// TIA Portal V16 program export: 2 tag tables, 6 data types, 3 data blocks, 4 code blocks (in call order from the OBs), 0 instance data blocks

VAR_GLOBAL   // PLC tag table "Default tag table"
END_VAR

VAR_GLOBAL   // PLC tag table "PAL_SystemTags"
   _SysSignals01 AT %MB0 : Byte;   // System signals byte 01 — Logic and scan synchronised pulses   {ExternalWritable false}
   _False AT %M0.0 : Bool;   // System Logic Bit — Always FALSE   {ExternalWritable false}
   _True AT %M0.1 : Bool;   // System Logic Bit — Always TRUE   {ExternalWritable false}
   _50ms AT %M0.2 : Bool;   // System Timing — 50 ms pulse scan synchronised   {ExternalWritable false}
   _100ms AT %M0.3 : Bool;   // System Timing — 100 ms pulse scan synchronised   {ExternalWritable false}
   _200ms AT %M0.4 : Bool;   // System Timing — 200 ms pulse scan synchronised   {ExternalWritable false}
   _500ms AT %M0.5 : Bool;   // System Timing — 500 ms pulse scan synchronised   {ExternalWritable false}
   _1s AT %M0.6 : Bool;   // System Timing — 1 s pulse scan synchronised   {ExternalWritable false}
   _2s AT %M0.7 : Bool;   // System Timing — 2 s pulse scan synchronised   {ExternalWritable false}
   _SysSignals02 AT %MB1 : Byte;   // System signals byte 02 — scan signals and common square waves   {ExternalWritable false}
   _CycleTick AT %M1.0 : Bool;   // System Timing — Cycle tick (active odd cycles, alternates with _CycleTock)   {ExternalWritable false}
   _CycleTock AT %M1.1 : Bool;   // System Timing — Cycle tock (active even cycles, alternates with _CycleTick)   {ExternalWritable false}
   _CycleFirst AT %M1.2 : Bool;   // System Timing — First cycle detected   {ExternalWritable false}
   _100msSqW AT %M1.3 : Bool;   // System Timing — 100 ms square wave scan synchronised   {ExternalWritable false}
   _200msSqW AT %M1.4 : Bool;   // System Timing — 200 ms square wave scan synchronised   {ExternalWritable false}
   _500msSqW AT %M1.5 : Bool;   // System Timing — 500 ms square wave scan synchronised   {ExternalWritable false}
   _1sSqW AT %M1.6 : Bool;   // System Timing — 1 s square wave scan synchronised   {ExternalWritable false}
   _2sSqW AT %M1.7 : Bool;   // System Timing — 2 s square wave scan synchronised   {ExternalWritable false}
   _ClockMem AT %MB10 : Byte;   // Clock Memory (populated by the CPU)   {ExternalWritable false}
   _ClockMem_100msSqW AT %M10.0 : Bool;   // Clock Memory — 10.0 Hz square wave 0.1 s period   {ExternalWritable false}
   _ClockMem_200msSqW AT %M10.1 : Bool;   // Clock Memory — 5.00 Hz square wave 0.2 s period   {ExternalWritable false}
   _ClockMem_400msSqW AT %M10.2 : Bool;   // Clock Memory — 2.50 Hz square wave 0.4 s period   {ExternalWritable false}
   _ClockMem_500msSqW AT %M10.3 : Bool;   // Clock Memory — 2.00 Hz square wave 0.5 s period   {ExternalWritable false}
   _ClockMem_800msSqW AT %M10.4 : Bool;   // Clock Memory — 1.25 Hz square wave 0.8 s period   {ExternalWritable false}
   _ClockMem_1000msSqW AT %M10.5 : Bool;   // Clock Memory — 1.00 Hz square wave 1.0 s period   {ExternalWritable false}
   _ClockMem_1600msSqW AT %M10.6 : Bool;   // Clock Memory — 0.62 Hz square wave 1.6 s period   {ExternalWritable false}
   _ClockMem_2000msSqW AT %M10.7 : Bool;   // Clock Memory — 0.50 Hz square wave 2.0 s period   {ExternalWritable false}
   _SysSignals AT %MW0 : Int;   // System signals   {ExternalWritable false}
END_VAR

TYPE "UT01000_St_SysRevision"
TITLE = Static UDT — Sys - Revision Data
// Revision Data
// stored: IsFailsafeCompliant false
   STRUCT
      REV_BLOCK { ExternalWritable := 'False'; S7_SetPoint := 'True'} : String[7];   // Block or Project number
      REV_NUMBER { ExternalWritable := 'False'; S7_SetPoint := 'True'} : String[20];   // Revision status followed by revision number
      REV_DATE { ExternalWritable := 'False'; S7_SetPoint := 'True'} : String[10];   // Revision date
      REV_AUTHOR { ExternalWritable := 'False'; S7_SetPoint := 'True'} : String[20];   // Revision author
   END_STRUCT;
END_TYPE

TYPE "UT01001_St_SysLicence"
TITLE = Static UDT — Sys - Licence Information
// Licence Information
// stored: IsFailsafeCompliant false
   STRUCT
      LICENCE_TYPE { ExternalWritable := 'False'} : String[20];   // Licence information — type of licence
      COPYRIGHT { ExternalWritable := 'False'} : String[30];   // Licence information — copyright (year and name)
   END_STRUCT;
END_TYPE

TYPE "UT21000_Dy_SysSignals"
TITLE = Dynamic UDT — Sys - Global Signals
// Global Logic and Timing Signals
// stored: IsFailsafeCompliant false
   STRUCT
      revInfo { ExternalWritable := 'False'} : "UT01000_St_SysRevision";   // ▀▀▀▀ UDT CURRENT REVISION
      ___________0010_0 { ExternalAccessible := 'False'; ExternalVisible := 'False'; ExternalWritable := 'False'} : Bool;
      ___________0010_1 { ExternalAccessible := 'False'; ExternalVisible := 'False'; ExternalWritable := 'False'} : Bool;   // ▀▀▀▀ SYSTEM SIGNALS
      _False { ExternalWritable := 'False'} : Bool;   // System Logic Bit — Always FALSE
      _True { ExternalWritable := 'False'} : Bool;   // System Logic Bit — Always TRUE
      _50ms { ExternalWritable := 'False'} : Bool;   // System Timing — 50 ms Pulse Scan synchronised
      _100ms { ExternalWritable := 'False'} : Bool;   // System Timing — 100 ms Pulse Scan synchronised
      _200ms { ExternalWritable := 'False'} : Bool;   // System Timing — 200 ms Pulse Scan synchronised
      _500ms { ExternalWritable := 'False'} : Bool;   // System Timing — 500 ms Pulse Scan synchronised
      _1s { ExternalWritable := 'False'} : Bool;   // System Timing — 1 s Pulse Scan synchronised
      _2s { ExternalWritable := 'False'} : Bool;   // System Timing — 2 s Pulse Scan synchronised
      _CycleTick { ExternalWritable := 'False'} : Bool;   // System Timing — Cycle tick (active odd cycles, alternates with _CycleTock)
      _CycleTock { ExternalWritable := 'False'} : Bool;   // System Timing — Cycle tock (active even cycles, alternates with _CycleTick)
      _CycleFirst { ExternalWritable := 'False'} : Bool;   // System Timing — First cycle detected
      _100msSqW { ExternalWritable := 'False'} : Bool;   // System Timing — 100 ms Square wave Scan synchronised
      _200msSqW { ExternalWritable := 'False'} : Bool;   // System Timing — 200 ms Square wave Scan synchronised
      _500msSqW { ExternalWritable := 'False'} : Bool;   // System Timing — 500 ms Square wave Scan synchronised
      _1sSqW { ExternalWritable := 'False'} : Bool;   // System Timing — 1 s Square wave Scan synchronised
      _2sSqW { ExternalWritable := 'False'} : Bool;   // System Timing — 2 s Square wave Scan synchronised
   END_STRUCT;
   // revInfo.REV_BLOCK := 'UT21000';
   // revInfo.REV_NUMBER := '000-801';
   // revInfo.REV_DATE := '2021-02-18';
   // revInfo.REV_AUTHOR := 'M. Gledhill';
END_TYPE

TYPE "UT21001_Dy_SysData"
TITLE = Dynamic UDT — Sys - Global Data
// Global System Data
// stored: IsFailsafeCompliant false
   STRUCT
      revInfo { ExternalWritable := 'False'} : "UT01000_St_SysRevision";   // ▀▀▀▀ UDT CURRENT REVISION
      ___________0010_0 { ExternalAccessible := 'False'; ExternalVisible := 'False'; ExternalWritable := 'False'} : Bool;
      ___________0010_1 { ExternalAccessible := 'False'; ExternalVisible := 'False'; ExternalWritable := 'False'} : Bool;   // ▀▀▀▀ CYCLE TIME DATA
      CycTime_Prev { ExternalWritable := 'False'} : Real;   // Previous cycle time (ms)
      CycTime_Max { ExternalWritable := 'False'} : Real;   // Maximum cycle time - since start-up (ms)
      CycTime_Min { ExternalWritable := 'False'} : Real;   // Minimum cycle time - since start-up (ms)
      Cyc_Counter { ExternalWritable := 'False'} : UDInt;   // Cycle rolling counter - incremented by 1 each scan
      __________0020_0 { ExternalAccessible := 'False'; ExternalVisible := 'False'; ExternalWritable := 'False'} : Bool := false;
      __________0020_1 { ExternalAccessible := 'False'; ExternalVisible := 'False'; ExternalWritable := 'False'} : Bool := false;   // ▀▀▀▀ REAL TIME CLOCK DATA
      RTC_Year { ExternalWritable := 'False'} : Int;   // Year (returns a value in the range 1970 to 2262)
      RTC_Month { ExternalWritable := 'False'} : Int;   // Month (1-12 representing Jan to Dec)
      RTC_Day { ExternalWritable := 'False'} : Int;   // Day of month (1-31)
      RTC_DayofWeek { ExternalWritable := 'False'} : Int;   // Day of week (1-7, where 1=Sunday, 7=Saturday)
      RTC_Hour { ExternalWritable := 'False'} : Int;   // Hour of day (0-23)
      RTC_Minute { ExternalWritable := 'False'} : Int;   // Minutes (0-59)
      RTC_Second { ExternalWritable := 'False'} : Int;   // Seconds (0-59)
      RTC_millisecond { ExternalWritable := 'False'} : Int;   // Milliseconds (0-999)
   END_STRUCT;
   // revInfo.REV_BLOCK := 'UT21001';
   // revInfo.REV_NUMBER := '001.000';
   // revInfo.REV_DATE := '2021-02-18';
   // revInfo.REV_AUTHOR := 'M. Gledhill ';
END_TYPE

TYPE "UT02001_St_InstAnalogRead"
TITLE = Static UDT — Inst - Analogue Instrument Read and Scale
// Analogue Instrument Read and Scale
// stored: IsFailsafeCompliant false
   STRUCT
      revInfo { ExternalWritable := 'False'} : "UT01000_St_SysRevision";   // Revision information
      ___________0010_0 { ExternalAccessible := 'False'; ExternalVisible := 'False'; ExternalWritable := 'False'} : Int;
      ___________0010_1 { ExternalAccessible := 'False'; ExternalVisible := 'False'; ExternalWritable := 'False'} : Int;   // ▀▀▀▀ INSTRUMENT CONFIGURATION
      CONFIG_ALM_H_ENABLE { ExternalWritable := 'False'; S7_SetPoint := 'True'} : Bool;   // CONFIG — High alarm is enabled (1 = enabled, 0 = no alarm)
      CONFIG_ALM_L_ENABLE { ExternalWritable := 'False'; S7_SetPoint := 'True'} : Bool;   // CONFIG — Low alarm is enabled (1 = enabled, 0 = no alarm)
      CONFIG_WRN_H_ENABLE { ExternalWritable := 'False'; S7_SetPoint := 'True'} : Bool;   // CONFIG — High warning is enabled (1 = enabled, 0 = no warning)
      CONFIG_WRN_L_ENABLE { ExternalWritable := 'False'; S7_SetPoint := 'True'} : Bool;   // CONFIG — Low warning is enabled (1 = enabled, 0 = no warning)
      CONFIG_FP_DISABLE { ExternalWritable := 'False'; S7_SetPoint := 'True'} : Bool;   // CONFIG — Faceplate is disabled (1 = no Faceplate, 0 = normal)
      CONFIG_SIM_DISABLE { ExternalWritable := 'False'; S7_SetPoint := 'True'} : Bool;   // CONFIG — Simulation is disabled (1 = no Simulation, 0 = normal)
      CONFIG_RL_ENABLE { ExternalWritable := 'False'; S7_SetPoint := 'True'} : Bool;   // CONFIG — Remote/local mode enabled (1 = remote/local permitted, 0 = remote/local N/A)
      ___________0020_0 { ExternalAccessible := 'False'; ExternalVisible := 'False'; ExternalWritable := 'False'} : Int;
      ___________0020_1 { ExternalAccessible := 'False'; ExternalVisible := 'False'; ExternalWritable := 'False'} : Int;   // ▀▀▀▀ INSTRUMENT RANGE & SCALING DATA
      RANGE_RAW_MIN { ExternalWritable := 'False'; S7_SetPoint := 'True'} : Int;   // RANGE — Minimum value of the raw analogue signal (at the card)
      RANGE_RAW_MAX { ExternalWritable := 'False'; S7_SetPoint := 'True'} : Int;   // RANGE — Maximum value of the raw analogue signal (at the card)
      RANGE_SCALE_MIN { ExternalWritable := 'False'; S7_SetPoint := 'True'} : Real;   // RANGE — Minimum value of the scaled analogue signal [engineering units]
      RANGE_SCALE_MAX { ExternalWritable := 'False'; S7_SetPoint := 'True'} : Real;   // RANGE — Maximum value of the scaled analogue signal [engineering units]
      RANGE_OOR_PERCENT { ExternalWritable := 'False'; S7_SetPoint := 'True'} : Real;   // RANGE — Out of range percentage (of raw range), beyond which the instrument is out of range
      ___________0030_0 { ExternalAccessible := 'False'; ExternalVisible := 'False'; ExternalWritable := 'False'} : Int;
      ___________0030_1 { ExternalAccessible := 'False'; ExternalVisible := 'False'; ExternalWritable := 'False'} : Int;   // ▀▀▀▀ INSTRUMENT INFORMATION (TAG & UNITS)
      INFO_TAG { ExternalWritable := 'False'; S7_SetPoint := 'True'} : String[20];   // INFORMATION — Instrument ID tag
      INFO_UNITS { ExternalWritable := 'False'; S7_SetPoint := 'True'} : String[10];   // INFORMATION — Engineering units of the instrument (unit of measure)
      ___________0040_0 { ExternalAccessible := 'False'; ExternalVisible := 'False'; ExternalWritable := 'False'} : Int;
      ___________0040_1 { ExternalAccessible := 'False'; ExternalVisible := 'False'; ExternalWritable := 'False'} : Int;   // ▀▀▀▀ INSTRUMENT ALARM/WARNING & HYSTERESIS SETPOINTS
      SP_ALM_H_VAL { ExternalWritable := 'False'; S7_SetPoint := 'True'} : Real;   // SETPOINT — High alarm threshold value [engineering units]
      SP_ALM_L_VAL { ExternalWritable := 'False'; S7_SetPoint := 'True'} : Real;   // SETPOINT — Low alarm threshold value [engineering units]
      SP_WRN_H_VAL { ExternalWritable := 'False'; S7_SetPoint := 'True'} : Real;   // SETPOINT — High warning threshold value [engineering units]
      SP_WRN_L_VAL { ExternalWritable := 'False'; S7_SetPoint := 'True'} : Real;   // SETPOINT — Low warning threshold value [engineering units]
      SP_ALM_H_HYST_VAL { ExternalWritable := 'False'; S7_SetPoint := 'True'} : Real;   // SETPOINT — High alarm hysteresis value [engineering units]
      SP_ALM_L_HYST_VAL { ExternalWritable := 'False'; S7_SetPoint := 'True'} : Real;   // SETPOINT — Low alarm hysteresis value [engineering units]
      SP_WRN_H_HYST_VAL { ExternalWritable := 'False'; S7_SetPoint := 'True'} : Real;   // SETPOINT — High warning hysteresis value [engineering units]
      SP_WRN_L_HYST_VAL { ExternalWritable := 'False'; S7_SetPoint := 'True'} : Real;   // SETPOINT — Low warning hysteresis value [engineering units]
      ___________0050_0 { ExternalAccessible := 'False'; ExternalVisible := 'False'; ExternalWritable := 'False'} : Int;
      ___________0050_1 { ExternalAccessible := 'False'; ExternalVisible := 'False'; ExternalWritable := 'False'} : Int;   // ▀▀▀▀ INSTRUMENT TIMER DEFAULT VALUES
      TIME_ALM_H_ON_DEL { ExternalWritable := 'False'; S7_SetPoint := 'True'} : Real;   // TIMER — High alarm on delay time (activation delay), [seconds]
      TIME_ALM_L_ON_DEL { ExternalWritable := 'False'; S7_SetPoint := 'True'} : Real;   // TIMER — Low alarm on delay time (activation delay), [seconds]
      TIME_WRN_H_ON_DEL { ExternalWritable := 'False'; S7_SetPoint := 'True'} : Real;   // TIMER — High warning on delay time (activation delay), [seconds]
      TIME_WRN_L_ON_DEL { ExternalWritable := 'False'; S7_SetPoint := 'True'} : Real;   // TIMER — Low warning on delay time (activation delay), [seconds]
      TIME_ALM_H_OFF_DEL { ExternalWritable := 'False'; S7_SetPoint := 'True'} : Real;   // TIMER — High alarm off delay time (deactivation delay), [seconds]
      TIME_ALM_L_OFF_DEL { ExternalWritable := 'False'; S7_SetPoint := 'True'} : Real;   // TIMER — Low alarm off delay time (deactivation delay), [seconds]
      TIME_WRN_H_OFF_DEL { ExternalWritable := 'False'; S7_SetPoint := 'True'} : Real;   // TIMER — High warning off delay time (deactivation delay), [seconds]
      TIME_WRN_L_OFF_DEL { ExternalWritable := 'False'; S7_SetPoint := 'True'} : Real;   // TIMER — Low warning off delay time (deactivation delay), [seconds]
   END_STRUCT;
   // revInfo.REV_BLOCK := 'UT02001';
   // revInfo.REV_NUMBER := '001.000';
   // revInfo.REV_DATE := '2021-02-18';
   // revInfo.REV_AUTHOR := 'M. Gledhill ';
END_TYPE

TYPE "UT22001_Dy_InstAnalogRead"
TITLE = Dynamic UDT — Inst - Analogue Instrument Read and Scale
// Analogue Instrument Read and Scale
// stored: IsFailsafeCompliant false
   STRUCT
      revInfo : "UT01000_St_SysRevision";   // Revision information
      ___________0010_0 { ExternalAccessible := 'False'; ExternalVisible := 'False'; ExternalWritable := 'False'} : Int;
      ___________0010_1 { ExternalAccessible := 'False'; ExternalVisible := 'False'; ExternalWritable := 'False'} : Int;   // ▀▀▀▀ STATUS (FOR BLOCK ICON AND SYMBOL)
      status_ConfigError : Bool;   // STATUS — Block is configured incorrectly
      status_Alm_H : Bool;   // STATUS — High alarm is active (1 = alarm active, 0 = no alarm)
      status_Alm_L : Bool;   // STATUS — Low alarm is active (1 = alarm active, 0 = no alarm)
      status_Wrn_H : Bool;   // STATUS — High warning is active (1 = warning active, 0 = no warning)
      status_Wrn_L : Bool;   // STATUS — Low warning is active (1 = warning active, 0 = no warning)
      status_Alm_H_Mask : Bool;   // STATUS — High alarm is masked (1 = alarm masked, 0 = normal)
      status_Alm_L_Mask : Bool;   // STATUS — Low alarm is masked (1 = alarm masked, 0 = normal)
      status_Wrn_H_Mask : Bool;   // STATUS — High warning is masked (1 = warning masked, 0 = normal)
      status_Wrn_L_Mask : Bool;   // STATUS — Low warning is masked (1 = warning masked, 0 = normal)
      status_Alm_H_Dis : Bool;   // STATUS — High alarm is disabled (1 = alarm disabled, 0 = normal)
      status_Alm_L_Dis : Bool;   // STATUS — Low alarm is disabled (1 = alarm disabled, 0 = normal)
      status_Wrn_H_Dis : Bool;   // STATUS — High warning is disabled (1 = warning disabled, 0 = normal)
      status_Wrn_L_Dis : Bool;   // STATUS — Low warning is disabled (1 = warning disabled, 0 = normal)
      status_Fault : Bool;   // STATUS — Instrument is in fault (1 = fault present, 0 = healthy)
      status_SimOn : Bool;   // STATUS — Instrument is in simulation mode (1 = simulation mode on, 0 = normal)
      status_RemoteOn : Bool;   // STATUS — Instrument is in remote mode (1 = remote mode, 0 = remote mode off)
      status_LocalOn : Bool;   // STATUS — Instrument is in local mode (1 = local mode, 0 = local mode off)
      status_RLOff : Bool;   // STATUS — Remote/local mode disabled (1 = ALL mode on, 0 = RL mode selected)
      ___________0020_0 { ExternalAccessible := 'False'; ExternalVisible := 'False'; ExternalWritable := 'False'} : Int;
      ___________0020_1 { ExternalAccessible := 'False'; ExternalVisible := 'False'; ExternalWritable := 'False'} : Int;   // ▀▀▀▀ OPERATING MODE SELECTION (FROM FACEPLATE OR PANEL)
      mode_Alm_H_MaskOn : Bool;   // MODE — Mask Alm_H (1 = mask alarm, 0 = normal)
      mode_Alm_L_MaskOn : Bool;   // MODE — Mask Alm_L (1 = mask alarm, 0 = normal)
      mode_Wrn_H_MaskOn : Bool;   // MODE — Mask Wrn_H (1 = mask warning, 0 = normal)
      mode_Wrn_L_MaskOn : Bool;   // MODE — Mask Wrn_H (1 = mask warning, 0 = normal)
      mode_SimOn : Bool;   // MODE — Simulation mode (1 = simulation mode active, 0 = normal)
      mode_SimValue : Real;   // MODE — Simulation value [engineering units]
      mode_LocalOn : Bool;   // MODE — Local HMI control enabled (1 = control active, 0 = control disabled or N/A)
      mode_RemoteOn : Bool;   // MODE — Remote SCADA control enabled (1 = control active, 0 = control disabled or N/A)
      ___________0030_0 { ExternalAccessible := 'False'; ExternalVisible := 'False'; ExternalWritable := 'False'} : Int;
      ___________0030_1 { ExternalAccessible := 'False'; ExternalVisible := 'False'; ExternalWritable := 'False'} : Int;   // ▀▀▀▀ MESSAGES (ALARMS, WARNINGS, FAULTS AND EVENTS)
      msg_Alm_H : Bool;   // MESSAGE — Alarm - high alarm is active
      msg_Alm_L : Bool;   // MESSAGE — Alarm - low alarm is active
      msg_Wrn_H : Bool;   // MESSAGE — Warning - high warning is active
      msg_Wrn_L : Bool;   // MESSAGE — Warning - low warning is active
      msg_Flt_External : Bool;   // MESSAGE — Fault - external fault signal is active
      msg_Flt_OverRange : Bool;   // MESSAGE — Fault - instrument is over-range
      msg_Flt_UnderRange : Bool;   // MESSAGE — Fault - instrument is under-range
      msg_Flt_OutOfRange : Bool;   // MESSAGE — Fault - instrument is out-of-range
      ___________0040_0 { ExternalAccessible := 'False'; ExternalVisible := 'False'; ExternalWritable := 'False'} : Int;
      ___________0040_1 { ExternalAccessible := 'False'; ExternalVisible := 'False'; ExternalWritable := 'False'} : Int;   // ▀▀▀▀ BATCH AND BOOKING DATA
      batch_ID : Int;   // BATCH — Booking ID (optional for batch operations)
      ___________0050_0 { ExternalAccessible := 'False'; ExternalVisible := 'False'; ExternalWritable := 'False'} : Int;
      ___________0050_1 { ExternalAccessible := 'False'; ExternalVisible := 'False'; ExternalWritable := 'False'} : Int;   // ▀▀▀▀ LIVE DATA (SCALED READING & TIMER VALUES)
      actual_Value : Real;   // ACTUAL — SCALED INSTRUMENT VALUE [engineering units]
      actual_Alm_H_Timer : Real;   // ACTUAL — Timer value — alarm high operation timer [seconds]
      actual_Alm_L_Timer : Real;   // ACTUAL — Timer value — alarm low operation timer [seconds]
      actual_Wrn_H_Timer : Real;   // ACTUAL — Timer value — warning high operation timer [seconds]
      actual_Wrn_L_Timer : Real;   // ACTUAL — Timer value — warning low operation timer [seconds]
      ___________0090_0 { ExternalAccessible := 'False'; ExternalVisible := 'False'; ExternalWritable := 'False'} : Int;
      ___________0090_1 { ExternalAccessible := 'False'; ExternalVisible := 'False'; ExternalWritable := 'False'} : Int;   // ▀▀▀▀ BLOCK INTERNAL WORKING AND STORAGE AREA
      "$pret_AlmHEn" : Bool;   // INTERNAL — Edge retention (+ve) alarm high enable
      "$Pret_AlmLEn" : Bool;   // INTERNAL — Edge retention (+ve) alarm low enable
      "$pret_WrnHEn" : Bool;   // INTERNAL — Edge retention (+ve) warning high enable
      "$pret_WrnLEn" : Bool;   // INTERNAL — Edge retention (+ve) warning low enable
   END_STRUCT;
   // revInfo.REV_BLOCK := 'UT22001';
   // revInfo.REV_NUMBER := '000.801';
   // revInfo.REV_DATE := '2021-02-18';
   // revInfo.REV_AUTHOR := 'M. Gledhill';
END_TYPE

DATA_BLOCK "DB21001_Dy_SysGlobalData"   // DB21001
TITLE = Dynamic DB — Sys - Global Data
{ S7_Optimized_Access := 'TRUE' }
AUTHOR : M_Gledhill
FAMILY : System
NAME : Dy_SysGlobalData
VERSION : 1.0
// PRACTICAL SERIES AUTOMATION LIBRARY (PAL)   —   COPYRIGHT 2020 – M. GLEDHILL (MIT LICENCE)
//                   ———— ◆ ————
//  FOR DETAILED DOCUMENTATION — SELECT THE BLOCK IN THE PROJECT TREE AND PRESS SHIFT + F1
//  FULL ONLINE DOCUMENTATION IS AVAILABLE AT: https://practicalseries.com/2001-pal/index.html
// stored: AutoNumber false, DBAccessibleFromOPCUA true, IsOnlyStoredInLoadMemory false, IsRetainMemResEnabled false, IsWriteProtectedInAS false, MemoryReserve 100
   VAR
      _DB_Header { ExternalWritable := 'False'} : Array[0..79] of Bool;   // STANDARD SYSTEM GLOBAL DATA
      __________0000_0 { ExternalWritable := 'False'} : Bool := false;
      __________0000_1 { ExternalWritable := 'False'} : Bool := false;   // ▀▀▀▀ DB CURRENT REVISION
      revInfo { ExternalWritable := 'False'} : "UT01000_St_SysRevision";
      __________0010_0 { ExternalWritable := 'False'} : Bool := false;
      __________0010_1 { ExternalWritable := 'False'} : Bool := false;   // ▀▀▀▀ PROJECT CURRENT REVISION
      projRevInfo { ExternalWritable := 'False'} : "UT01000_St_SysRevision";
      __________0020_0 { ExternalWritable := 'False'} : Bool := false;
      __________0020_1 { ExternalWritable := 'False'} : Bool := false;   // ▀▀▀▀ SYSTEM SIGNALS — LOGIC AND TIMING SIGNALS
      SysSignals { ExternalWritable := 'False'} : "UT21000_Dy_SysSignals";
      __________0030_0 { ExternalWritable := 'False'} : Bool := false;
      __________0030_1 { ExternalWritable := 'False'} : Bool := false;   // ▀▀▀▀ SYSTEM DATA — CYCLE TIMING AND RTC
      SysData { ExternalWritable := 'False'} : "UT21001_Dy_SysData";
      __________0040_0 { ExternalWritable := 'False'} : Bool := false;
      __________0040_1 { ExternalWritable := 'False'} : Bool := false;   // ▀▀▀▀ OB CALL TIMES
      OB10_CallTime { ExternalWritable := 'False'} : DTL;   // Time of day interrupt 1
      OB11_CallTime { ExternalWritable := 'False'} : DTL;   // Time of day interrupt 2
      OB12_CallTime { ExternalWritable := 'False'} : DTL;   // Time of day interrupt 3
      OB13_CallTime { ExternalWritable := 'False'} : DTL;   // Time of day interrupt 4
      OB14_CallTime { ExternalWritable := 'False'} : DTL;   // Time of day interrupt 5
      OB15_CallTime { ExternalWritable := 'False'} : DTL;   // Time of day interrupt 6
      OB16_CallTime { ExternalWritable := 'False'} : DTL;   // Time of day interrupt 7
      OB17_CallTime { ExternalWritable := 'False'} : DTL;   // Time of day interrupt 8
      OB20_CallTime { ExternalWritable := 'False'} : DTL;   // Time delay interrupt 1
      OB21_CallTime { ExternalWritable := 'False'} : DTL;   // Time delay interrupt 2
      OB22_CallTime { ExternalWritable := 'False'} : DTL;   // Time delay interrupt 3
      OB23_CallTime { ExternalWritable := 'False'} : DTL;   // Time delay interrupt 4
      OB30_CallTime { ExternalWritable := 'False'} : DTL;   // Timed cyclic interrupt 1
      OB31_CallTime { ExternalWritable := 'False'} : DTL;   // Timed cyclic interrupt 2
      OB32_CallTime { ExternalWritable := 'False'} : DTL;   // Timed cyclic interrupt 3
      OB33_CallTime { ExternalWritable := 'False'} : DTL;   // Timed cyclic interrupt 4
      OB34_CallTime { ExternalWritable := 'False'} : DTL;   // Timed cyclic interrupt 5
      OB35_CallTime { ExternalWritable := 'False'} : DTL;   // Timed cyclic interrupt 6
      OB36_CallTime { ExternalWritable := 'False'} : DTL;   // Timed cyclic interrupt 7
      OB37_CallTime { ExternalWritable := 'False'} : DTL;   // Timed cyclic interrupt 8
      OB38_CallTime { ExternalWritable := 'False'} : DTL;   // Timed cyclic interrupt 9
      OB40_CallTime { ExternalWritable := 'False'} : DTL;   // Hardware interrupt 1
      OB41_CallTime { ExternalWritable := 'False'} : DTL;   // Hardware interrupt 2
      OB42_CallTime { ExternalWritable := 'False'} : DTL;   // Hardware interrupt 3
      OB43_CallTime { ExternalWritable := 'False'} : DTL;   // Hardware interrupt 4
      OB44_CallTime { ExternalWritable := 'False'} : DTL;   // Hardware interrupt 5
      OB45_CallTime { ExternalWritable := 'False'} : DTL;   // Hardware interrupt 6
      OB46_CallTime { ExternalWritable := 'False'} : DTL;   // Hardware interrupt 7
      OB47_CallTime { ExternalWritable := 'False'} : DTL;   // Hardware interrupt 8
      OB80_CallTime { ExternalWritable := 'False'} : DTL;   // Error interrupt — max cycle time exceeded
      OB82_CallTime { ExternalWritable := 'False'} : DTL;   // Error interrupt — module diagnostic
      OB83_CallTime { ExternalWritable := 'False'} : DTL;   // Error interrupt — module changed
      OB86_CallTime { ExternalWritable := 'False'} : DTL;   // Error interrupt — rack fault
      OB100_CallTime { ExternalWritable := 'False'} : DTL;   // Start-up interrupt
      OB121_CallTime { ExternalWritable := 'False'} : DTL;   // Error interrupt — programming fault
      OB122_CallTime { ExternalWritable := 'False'} : DTL;   // Error interrupt — IO access fault
   END_VAR
BEGIN
   // _DB_Header[0] : ▀▀▀▀▀▀▀▀▀▀▀▀▀▀▀▀▀▀▀▀▀▀▀▀▀▀▀▀▀▀▀▀▀▀▀▀▀▀▀▀▀▀▀▀
   // _DB_Header[2] : TITLE: STANDARD SYSTEM GLOBAL DATA
   // _DB_Header[4] : ▄▄▄▄▄▄▄▄▄▄▄▄▄▄▄▄▄▄▄▄▄▄▄▄▄▄▄▄▄▄▄▄▄▄▄▄▄▄▄▄▄▄▄▄
   // _DB_Header[5] : TYPE: DYNAMIC
   // _DB_Header[6] : ▀▀▀▀▀▀▀▀▀▀▀▀▀▀▀▀▀▀▀▀▀▀▀▀▀▀▀▀▀▀▀▀▀▀▀▀▀▀▀▀▀▀▀▀
   // _DB_Header[8] : Global system data storage DB. The block records various system variables and information:
   // _DB_Header[10] : • Project revision data
   // _DB_Header[11] : • Common system signals (logic and timing)
   // _DB_Header[12] : • Cycle timing information (previous, max, min and a cycle counter)
   // _DB_Header[13] : • CPU real time clock data (in globally readable format)
   // _DB_Header[14] : • Last call time of any interrupt OB
   // _DB_Header[16] : The cycle timing information and the RTC data are provided by FC01000. The interrupt OB data
   // _DB_Header[17] : is provided by the individual OBs.
   // _DB_Header[19] : ━━━ ⬙⬙⬙⬙⬙⬙ ━━━
   // _DB_Header[21] : ▄▄▄▄▄▄▄▄▄▄▄▄▄▄▄▄▄▄▄▄▄▄▄▄▄▄▄▄▄▄▄▄▄▄▄▄▄▄▄▄▄▄▄▄
   // _DB_Header[22] : MODIFICATION HISTORY
   // _DB_Header[24] : This is a summary of the recent software modifications made to this block (most recent at top)
   // _DB_Header[26] : ―――――――――――――――――――――――――――――――――――――――――――
   // _DB_Header[27] : DATE REVISION MASTER BRANCH DEV
   // _DB_Header[28] : (nnn.amm) COMMIT TAG (Base ---> Merge) BRANCH Author
   // _DB_Header[29] : ———————————————————————————————————————————
   // _DB_Header[30] : 2020.11.18 001.000 D0002A-001.000 D0002 D0003 D0002A M. Gledhill
   // _DB_Header[31] : FC01001 Migration to VCS — Released for use
   // _DB_Header[32] : 2020.11.18 000.801 D0002A-000.801 D0002 N/A D0002A M. Gledhill
   // _DB_Header[33] : FC01001 Migration to VCS — Released for test
   // _DB_Header[34] : ———————————————————————————————————————————
   // _DB_Header[35] : Where: nnn = Major revision
   // _DB_Header[36] : a = Type (1-7 Development, 8 Proving, 9 Qualification, 0 Release)
   // _DB_Header[37] : mm = Minor revision (must be 00 if a = 0)
   // _DB_Header[38] : Block properties version number should be set to nn.a (only one decimal place)
   // _DB_Header[40] : ██████████████ █ █ █ █ END █ █ █ █ ██████████████
   revInfo.REV_BLOCK := 'DB21001';
   revInfo.REV_NUMBER := '001.000';
   revInfo.REV_DATE := '2021-02-18';
   revInfo.REV_AUTHOR := 'M. Gledhill';
END_DATA_BLOCK

DATA_BLOCK "DB02001_St_InstAnalogRead"   // DB2001
TITLE = Static DB — Inst - Analogue Instrument Read and Scale
{ S7_Optimized_Access := 'TRUE' }
AUTHOR : M_Gledhill
FAMILY : Instrumentation
NAME : St_InstAnalogRead
VERSION : 1.0
// PRACTICAL SERIES AUTOMATION LIBRARY (PAL)   —   COPYRIGHT 2020 – M. GLEDHILL (MIT LICENCE)
//                   ———— ◆ ————
//  FOR DETAILED DOCUMENTATION — SELECT THE BLOCK IN THE PROJECT TREE AND PRESS SHIFT + F1
//  FULL ONLINE DOCUMENTATION IS AVAILABLE AT: https://practicalseries.com/2001-pal/index.html
// stored: AutoNumber false, DBAccessibleFromOPCUA true, IsOnlyStoredInLoadMemory false, IsRetainMemResEnabled false, IsWriteProtectedInAS false, MemoryReserve 100
   VAR
      _DB_Header { ExternalAccessible := 'False'; ExternalVisible := 'False'; ExternalWritable := 'False'} : Array[0..79] of Bool;   // STANDARD ANALOGUE INSTRUMENT READ
      __________0000_0 { ExternalAccessible := 'False'; ExternalVisible := 'False'; ExternalWritable := 'False'} : Bool := false;
      __________0000_1 { ExternalAccessible := 'False'; ExternalVisible := 'False'; ExternalWritable := 'False'} : Bool := false;   // ▀▀▀▀ DB CURRENT REVISION
      revInfo { ExternalWritable := 'False'; S7_SetPoint := 'True'} : "UT01000_St_SysRevision";
      __________0010_0 { ExternalAccessible := 'False'; ExternalVisible := 'False'; ExternalWritable := 'False'} : Bool := false;
      __________0010_1 { ExternalAccessible := 'False'; ExternalVisible := 'False'; ExternalWritable := 'False'} : Bool := false;   // ▀▀▀▀ ANALOGUE INSTRUMENTS
      FIC101 { ExternalWritable := 'False'; S7_SetPoint := 'True'} : "UT02001_St_InstAnalogRead";   // Filter 1 outlet flow
   END_VAR
BEGIN
   // _DB_Header[0] : ▀▀▀▀▀▀▀▀▀▀▀▀▀▀▀▀▀▀▀▀▀▀▀▀▀▀▀▀▀▀▀▀▀▀▀▀▀▀▀▀▀▀▀▀
   // _DB_Header[2] : TITLE: STANDARD ANALOGUE INSTRUMENT READ (SCALE & ALARM MONITORING)
   // _DB_Header[4] : ▄▄▄▄▄▄▄▄▄▄▄▄▄▄▄▄▄▄▄▄▄▄▄▄▄▄▄▄▄▄▄▄▄▄▄▄▄▄▄▄▄▄▄▄
   // _DB_Header[5] : TYPE: STATIC
   // _DB_Header[6] : ▀▀▀▀▀▀▀▀▀▀▀▀▀▀▀▀▀▀▀▀▀▀▀▀▀▀▀▀▀▀▀▀▀▀▀▀▀▀▀▀▀▀▀▀
   // _DB_Header[8] : This is the static data block associated with the standard analogue instrument read
   // _DB_Header[9] : block:
   // _DB_Header[10] : FC02001_StdInstAnalogRead
   // _DB_Header[12] : The static data holds the threshold values for any configured alarms and warnings,
   // _DB_Header[13] : activation delays, scaled and raw value ranges and various configuration options.
   // _DB_Header[15] : Each instrument is given the user data type:
   // _DB_Header[16] : UT02001_St_InstAnalogueRead
   // _DB_Header[17] : This holds the full set of static configuration data for the instrument.
   // _DB_Header[19] : ━━━ ⬙⬙⬙⬙⬙⬙ ━━━
   // _DB_Header[21] : ▄▄▄▄▄▄▄▄▄▄▄▄▄▄▄▄▄▄▄▄▄▄▄▄▄▄▄▄▄▄▄▄▄▄▄▄▄▄▄▄▄▄▄▄
   // _DB_Header[22] : MODIFICATION HISTORY
   // _DB_Header[24] : This is a summary of the recent software modifications made to this block (most recent at top)
   // _DB_Header[26] : ―――――――――――――――――――――――――――――――――――――――――――
   // _DB_Header[27] : DATE REVISION MASTER BRANCH DEV
   // _DB_Header[28] : (nnn.amm) COMMIT TAG (Base ---> Merge) BRANCH Author
   // _DB_Header[29] : ———————————————————————————————————————————
   // _DB_Header[30] : 2020.11.18 000.801 D0002B-000.801 D0002 N/A D0002B M. Gledhill
   // _DB_Header[31] : FC02001 Migration to VCS — Released for test
   // _DB_Header[32] : ———————————————————————————————————————————
   // _DB_Header[33] : Where: nnn = Major revision
   // _DB_Header[34] : a = Type (1-7 Development, 8 Proving, 9 Qualification, 0 Release)
   // _DB_Header[35] : mm = Minor revision (must be 00 if a = 0)
   // _DB_Header[36] : Block properties version number should be set to nn.a (only one decimal place)
   // _DB_Header[38] : ██████████████ █ █ █ █ END █ █ █ █ ██████████████
   revInfo.REV_BLOCK := 'DB02001';
   revInfo.REV_NUMBER := '000.801';
   revInfo.REV_DATE := '2021-02-18';
   revInfo.REV_AUTHOR := 'M. Gledhill';
   FIC101.CONFIG_ALM_H_ENABLE := true;
   FIC101.CONFIG_ALM_L_ENABLE := true;
   FIC101.CONFIG_WRN_H_ENABLE := true;
   FIC101.CONFIG_WRN_L_ENABLE := true;
   FIC101.CONFIG_FP_DISABLE := false;
   FIC101.CONFIG_SIM_DISABLE := false;
   FIC101.CONFIG_RL_ENABLE := false;
   FIC101.RANGE_RAW_MAX := 27648;
   FIC101.RANGE_SCALE_MIN := 0.0;
   FIC101.RANGE_SCALE_MAX := 1000.0;
   FIC101.RANGE_OOR_PERCENT := 2.5;
   FIC101.INFO_TAG := 'FIC101';
   FIC101.INFO_UNITS := 'l/s';
   FIC101.SP_ALM_H_VAL := 750.0;
   FIC101.SP_ALM_L_VAL := 250.0;
   FIC101.SP_WRN_H_VAL := 625.0;
   FIC101.SP_WRN_L_VAL := 375.0;
   FIC101.SP_ALM_H_HYST_VAL := 62.5;
   FIC101.SP_ALM_L_HYST_VAL := 62.0;
   FIC101.SP_WRN_H_HYST_VAL := 61.5;
   FIC101.SP_WRN_L_HYST_VAL := 61.0;
   FIC101.TIME_ALM_H_ON_DEL := 10.0;
   FIC101.TIME_ALM_L_ON_DEL := 11.0;
   FIC101.TIME_WRN_H_ON_DEL := 12.0;
   FIC101.TIME_WRN_L_ON_DEL := 13.0;
   FIC101.TIME_ALM_H_OFF_DEL := 15.0;
   FIC101.TIME_ALM_L_OFF_DEL := 16.0;
   FIC101.TIME_WRN_H_OFF_DEL := 17.0;
   FIC101.TIME_WRN_L_OFF_DEL := 18.0;
END_DATA_BLOCK

DATA_BLOCK "DB22001_Dy_InstAnalogRead"   // DB22001
TITLE = Dynamic DB — Inst - Analogue Instrument Read and Scale
{ S7_Optimized_Access := 'TRUE' }
AUTHOR : M_Gledhill
FAMILY : Instrumentation
NAME : Dy_InstAnalogRead
VERSION : 1.0
// PRACTICAL SERIES AUTOMATION LIBRARY (PAL)   —   COPYRIGHT 2018 – M. GLEDHILL (MIT LICENCE)
//                   ———— ◆ ————
//  FOR DETAILED DOCUMENTATION — SELECT THE BLOCK IN THE PROJECT TREE AND PRESS SHIFT + F1
//  FULL ONLINE DOCUMENTATION IS AVAILABLE AT: https://practicalseries.com/2001-pal/index.html
// stored: AutoNumber false, DBAccessibleFromOPCUA true, IsOnlyStoredInLoadMemory false, IsRetainMemResEnabled false, IsWriteProtectedInAS false, MemoryReserve 100
   VAR
      _DB_Header { ExternalAccessible := 'False'; ExternalVisible := 'False'; ExternalWritable := 'False'} : Array[0..79] of Bool;   // STANDARD ANALOGUE INSTRUMENT READ
      __________0000_0 { ExternalAccessible := 'False'; ExternalVisible := 'False'; ExternalWritable := 'False'} : Bool := false;
      __________0000_1 { ExternalAccessible := 'False'; ExternalVisible := 'False'; ExternalWritable := 'False'} : Bool := false;   // ▀▀▀▀ DB CURRENT REVISION
      revInfo { ExternalWritable := 'False'; S7_SetPoint := 'True'} : "UT01000_St_SysRevision";
      __________0010_0 { ExternalAccessible := 'False'; ExternalVisible := 'False'; ExternalWritable := 'False'} : Bool := false;
      __________0010_1 { ExternalAccessible := 'False'; ExternalVisible := 'False'; ExternalWritable := 'False'} : Bool := false;   // ▀▀▀▀ ANALOGUE INSTRUMENTS
      FIC101 { S7_SetPoint := 'True'} : "UT22001_Dy_InstAnalogRead";   // Filter 1 outlet flow
   END_VAR
BEGIN
   // _DB_Header[0] : ▀▀▀▀▀▀▀▀▀▀▀▀▀▀▀▀▀▀▀▀▀▀▀▀▀▀▀▀▀▀▀▀▀▀▀▀▀▀▀▀▀▀▀▀
   // _DB_Header[2] : TITLE: STANDARD ANALOGUE INSTRUMENT READ (SCALE & ALARM MONITORING)
   // _DB_Header[4] : ▄▄▄▄▄▄▄▄▄▄▄▄▄▄▄▄▄▄▄▄▄▄▄▄▄▄▄▄▄▄▄▄▄▄▄▄▄▄▄▄▄▄▄▄
   // _DB_Header[5] : TYPE: DYNAMIC
   // _DB_Header[6] : ▀▀▀▀▀▀▀▀▀▀▀▀▀▀▀▀▀▀▀▀▀▀▀▀▀▀▀▀▀▀▀▀▀▀▀▀▀▀▀▀▀▀▀▀
   // _DB_Header[8] : This is the dynamic data block associated with the standard analogue instrument read
   // _DB_Header[9] : block:
   // _DB_Header[10] : FC02001_StdInstAnalog
   // _DB_Header[12] : The dynamic data holds the current scaled value of the instrument, along with
   // _DB_Header[13] : any alarms, warnings or faults.
   // _DB_Header[15] : Each instrument is given the user data type:
   // _DB_Header[16] : UT22001_Dy_InstAnalogue
   // _DB_Header[17] : This holds the full set of static configuration data for the instrument.
   // _DB_Header[19] : ━━━ ⬙⬙⬙⬙⬙⬙ ━━━
   // _DB_Header[21] : ▄▄▄▄▄▄▄▄▄▄▄▄▄▄▄▄▄▄▄▄▄▄▄▄▄▄▄▄▄▄▄▄▄▄▄▄▄▄▄▄▄▄▄▄
   // _DB_Header[22] : MODIFICATION HISTORY
   // _DB_Header[24] : This is a summary of the recent software modifications made to this block (most recent at top)
   // _DB_Header[26] : ―――――――――――――――――――――――――――――――――――――――――――
   // _DB_Header[27] : DATE REVISION MASTER BRANCH DEV
   // _DB_Header[28] : (nnn.amm) COMMIT TAG (Base ---> Merge) BRANCH Author
   // _DB_Header[29] : ———————————————————————————————————————————
   // _DB_Header[30] : 2020.11.18 001.000 D0002B-001.000 D0002 D0004 D0002B M. Gledhill
   // _DB_Header[31] : FC02001 Migration to VCS — Released for use
   // _DB_Header[32] : 2020.11.18 000.801 D0002B-000.801 D0002 N/A D0002B M. Gledhill
   // _DB_Header[33] : FC02001 Migration to VCS — Released for test
   // _DB_Header[34] : ———————————————————————————————————————————
   // _DB_Header[35] : Where: nnn = Major revision
   // _DB_Header[36] : a = Type (1-7 Development, 8 Proving, 9 Qualification, 0 Release)
   // _DB_Header[37] : mm = Minor revision (must be 00 if a = 0)
   // _DB_Header[38] : Block properties version number should be set to nn.a (only one decimal place)
   // _DB_Header[40] : ██████████████ █ █ █ █ END █ █ █ █ ██████████████
   revInfo.REV_BLOCK := 'DB22001';
   revInfo.REV_NUMBER := '001.000';
   revInfo.REV_DATE := '2021-02-18';
   revInfo.REV_AUTHOR := 'M. Gledhill';
END_DATA_BLOCK

ORGANIZATION_BLOCK "OB00001_IntNMainProgram"   // OB1, LAD, ProgramCycle
TITLE = Interrupt - Norm — Main Program Cyclic Execution
{ S7_Optimized_Access := 'TRUE' }
AUTHOR : M_Gledhill
FAMILY : Interrupt
NAME : IntNMainProgram
VERSION : 0.0.0.0
// PRACTICAL SERIES AUTOMATION LIBRARY (PAL)   —   COPYRIGHT 2020 – M. GLEDHILL (MIT LICENCE)
//                   ———— ◆ ————
//  FOR DETAILED DOCUMENTATION — SELECT THE BLOCK IN THE PROJECT TREE AND PRESS SHIFT + F1
//  FULL ONLINE DOCUMENTATION IS AVAILABLE AT: https://practicalseries.com/2001-pal/index.html
// stored: AutoNumber true, IsIECCheckEnabled false, SetENOAutomatically false
   VAR_INPUT
      Initial_Call : Bool;   // Initial call of this OB
      Remanence : Bool;   // =True, if remanent data are available
   END_VAR
   VAR_TEMP
      revInfo : "UT01000_St_SysRevision";   // Revision information for this block
      licInfo : "UT01001_St_SysLicence";   // Licence information for this block
   END_VAR
BEGIN

REGION Network 1: Project description
   // ▀▀▀▀▀▀▀▀▀▀▀▀▀▀▀▀▀▀▀▀▀▀▀▀▀▀▀▀▀▀▀▀▀▀▀▀▀▀▀▀▀▀▀▀
   // 
   // TITLE:    PS2001 — PRACTICAL SERIES AUTOMATION LIBRARY
   // 
   // ▄▄▄▄▄▄▄▄▄▄▄▄▄▄▄▄▄▄▄▄▄▄▄▄▄▄▄▄▄▄▄▄▄▄▄▄▄▄▄▄▄▄▄▄
   // 
   // 
   // ――――――――――――――――――――――――――――――――――
   // COPYRIGHT:       © 2020 Michael Gledhill
   //           Part of the Practical Series of Publications
   //           Published in the United Kingdom
   //           mg@practicalseries.com
   //           https://practicalseries.com
   // ――――――――――――――――――――――――――――――――――
   // CUSTOMER:       Practical Series of Publications (PSP)
   // 
   // PROJECT:      Practical Series Automation Library (PAL)
   // 
   // PROJECT NO.:       PS2001
   // ――――――――――――――――――――――――――――――――――
   // CONTROLLER:       CPU 1515-2PN/DP
   // 
   // CONTROLLER NAME:    CON100
   // 
   // IP ADDRESS:      192.168.001.100
   // ――――――――――――――――――――――――――――――――――
   // TIA PROJECT NAME:    PS2001-VCS-D0002 — BASELINE BUILD
   // 
   // STATUS:        DEVELOPMENT
   // ――――――――――――――――――――――――――――――――――
   // PROTECTION:     To minimise the risk of inadvertent modification to 
   //           tested modules, certain blocks will be released for 
   //           use with “protected access” (referred to a “write 
   //           protection” in Siemens terminology), this allows the 
   //           block to be used normally, but prevents the block 
   //           being accidentally modified. 
   // 
   //           This is in accordance with the risk assessment given 
   //           in the Validation Plant (VP), Appendix A [Ref. 002].
   // 
   //           ┌─────────────────────┐
   //           │ THE WRITE PROTECTION PASSWORD IS: PS2001 │
   //           └─────────────────────┘
   // 
   // 
   // ▄▄▄▄▄▄▄▄▄▄▄▄▄▄▄▄▄▄▄▄▄▄▄▄▄▄▄▄▄▄▄▄▄▄▄▄▄▄▄▄▄▄▄▄
   // PROJECT OVERVIEW
   // 
   // 
   // The PAL is a library of software modules and templates that have been developed for the 
   // Siemens Simatic S7-1500 range of controllers (and to a lesser extent the S7-1200 range).
   // 
   // The full library and all necessary documentation is available from the Practical Series website:
   // 
   //      https://practicalseries.com/2001-pal/index.html
   // 
   // 
   // The PAL is configured and deployed using the Siemens Simatic TIA Portal programming 
   // environment.
   // 
   // The PAL software structure is designed such that it is applicable to virtually all industrial 
   // applications that can generally controlled by a programmable logic controller.
   // 
   // The PAL software being developed as part of this Project, is considered to be suitable for use in 
   // the following types of industries (this is not an exhaustive list):
   // 
   //    •   Water and waste water treatment
   //    •   Pharmaceutical and batch production
   //    •   Brewing and fermentation
   //    •   Chemical manufacturing
   //    •   Oil and gas systems
   //    •   Food and beverage production
   // 
   // Such applications can generally be thought of as processes that operate with a response time
   // of more than 100 ms. I.e. the system would not be expected to respond to some stimuli faster
   // than 100 ms. In practice, a Controller may (and usually will) respond faster than this; however, 
   // a response time of 100 ms is considered to be an acceptable limit for PLC control.
   // 
   // At its most basic level, the PAL will be a library of software modules that control the fundamental 
   // aspects of an industrial plant; such modules would for example read the value of an instrument, 
   // operate a valve or drive, perform a calculation &c.
   // 
   // Such software modules are referred to as standard modules, these are fixed modules that 
   // perform a particular function and are identical across all software installations.
   // 
   // The PAL also contains application specific modules; these contain software that is applicable 
   // to the plant being controlled.
   // 
   // The Practical Series Automation Library is freely available under the MIT Open Source licence 
   // (see below). Those who find it useful may, if they wish, make a donation to support the library. 
   // 
   // Donations can be made here:
   // 
   //      https://practicalseries.com/2001-pal/11-web/81-00-pay.html
   // 
   // The PAL contains fully deployable software that has been developed by the author in his 
   // profession as a chartered electrical engineer. It is currently in use on various live plants 
   // throughout the UK and in some other parts of the world. 
   // 
   // This software is suitable for controlling and automating most industrial applications (typical 
   // process applications). It is easy to use and configure, but does have a degree of practical 
   // complexity appropriate for the environments within which it is employed. It is heavily 
   // configurable, has various operating modes and is suitable for a multitude of industrial 
   // applications.
   // 
   // IF YOU DON’T UNDERSTAND IT, DON’T USE IT. IF YOU DO USE IT, YOU DO SO AT YOUR OWN RISK.
   // 
   //                ━━━   ⬙⬙⬙⬙⬙⬙   ━━━
   // 
   // ▄▄▄▄▄▄▄▄▄▄▄▄▄▄▄▄▄▄▄▄▄▄▄▄▄▄▄▄▄▄▄▄▄▄▄▄▄▄▄▄▄▄▄▄
   // DOCUMENT REFERENCES
   // 
   //  ――――――――――――――――――――――――――――――――――――――――――
   //  REF.     DOCUMENT NO.       TITLE
   //  ――――――――――――――――――――――――――――――――――――――――――
   //  001  PS2001-5-0101-001   Quality Plan (QP)
   //  002  PS2001-5-0121-002   Validation Plan (VP)
   //  003  PS2001-5-0131-003   Test Plan (TP)
   //  004  PS2001-5-1101-001   User requirements specification (URS)
   //  005  PS2001-5-1111-001   Requirement Traceability Matrix (RTM)
   //  006  PS2001-5-2101-001   Functional Specification (FS) 
   //  007  PS2001-5-2211-001   Hardware Design Specification (HDS)
   //  008  PS2001-5-2311-001   Software Design Specification (SDS)
   //  009  PS2001-5-7111-001   User Guide (UG)
   //  010  PS2001-5-2313-011   Style Guide (SG)
   //  011  PS2001-5-2312-fcNo.    Software Module Design Specification (SMDS)
   //  012  PS2001-5-2301-001   Software Module Register (SMR)
   //  013  PS2001-5-2302-011   Software Control and Mechanism (SCM)
   //  ――――――――――――――――――――――――――――――――――――――――――
   // 
   //                ━━━   ⬙⬙⬙⬙⬙⬙   ━━━
   // 
   // 
   // ▄▄▄▄▄▄▄▄▄▄▄▄▄▄▄▄▄▄▄▄▄▄▄▄▄▄▄▄▄▄▄▄▄▄▄▄▄▄▄▄▄▄▄▄
   // COMPLETED MODULES 
   // 
   //  ――――――――――――――――――――-―-- STATIC DATA       ― DYNAMIC  DAT A   ―
   //  BLOCK     NAME         REVISION    UDT/DB    REVISION  UDT/DB    REVISION  
   //  ――――――――――――――――――――――――――――――――――――――――――
   //  FC61000 DocGenExample     001.000   None           None 
   //                  2021.02.18   None           None          
   //  ――――――――――――――――――――――――――――――――――――――――――
   //  See Software Module Register [Ref. 012] for full details
   // 
   //                ━━━   ⬙⬙⬙⬙⬙⬙   ━━━
   // 
   // 
   // ▀▀▀▀▀▀▀▀▀▀▀▀▀▀▀▀▀▀▀▀▀▀▀▀▀▀▀▀▀▀▀▀▀▀▀▀▀▀▀▀▀▀▀▀
   // LICENCE AND CONTACT INFORMATION
   // 
   // This software and its associated documentation is made available under the MIT Licence:
   // 
   // ════════════════════════════════════════════
   // 
   // The MIT License (MIT)
   // 
   // Copyright © 2020 Michael Gledhill
   // 
   // Permission is hereby granted, free of charge, to any person obtaining a copy of this software 
   // and associated documentation files (the “Software”), to deal in the Software without restriction, 
   // including without limitation the rights to use, copy, modify, merge, publish, distribute, 
   // sublicense, and/or sell copies of the Software, and to permit persons to whom the Software is 
   // furnished to do so, subject to the following conditions: 
   // 
   // The above copyright notice and this permission notice shall be included in all copies or 
   // substantial portions of the Software.
   // 
   // THE SOFTWARE IS PROVIDED “AS IS”, WITHOUT WARRANTY OF ANY KIND, EXPRESS OR IMPLIED, 
   // INCLUDING BUT NOT LIMITED TO THE WARRANTIES OF MERCHANTABILITY, FITNESS FOR A 
   // PARTICULAR PURPOSE AND NON-INFRINGEMENT. IN NO EVENT SHALL THE AUTHORS OR COPYRIGHT 
   // HOLDERS BE LIABLE FOR ANY CLAIM, DAMAGES OR OTHER LIABILITY, WHETHER IN AN ACTION OF 
   // CONTRACT, TORT OR OTHERWISE, ARISING FROM, OUT OF OR IN CONNECTION WITH THE SOFTWARE 
   // OR THE USE OR OTHER DEALINGS IN THE SOFTWARE.
   // 
   // ════════════════════════════════════════════
   //                    ┌────────────┐
   // You can reach the author by email here:   │  mg@practicalseries.com  │
   //                    └────────────┘
   // Questions, corrections, constructive criticism and complaints (polite ones) are invited.
   // 
   // ▄▄▄▄▄▄▄▄▄▄▄▄▄▄▄▄▄▄▄▄▄▄▄▄▄▄▄▄▄▄▄▄▄▄▄▄▄▄▄▄▄▄▄▄
   // 
   // 
   //                ━━━   ⬙⬙⬙⬙⬙⬙   ━━━
   // 
   // 
   // 
   // ██████████████ █ █ █ █  END   █ █ █ █ ██████████████
END_REGION

REGION Network 2: Current revision and modification history
   // ▄▄▄▄▄▄▄▄▄▄▄▄▄▄▄▄▄▄▄▄▄▄▄▄▄▄▄▄▄▄▄▄▄▄▄▄▄▄▄▄▄▄▄▄
   // MODIFICATION HISTORY
   // 
   // The revision data shown here, in the network comments, contains additional information 
   // reflecting the software development workflow under the version control system (VCS) employed 
   // to track all software changes.
   // 
   // The VCS in use is the Git Source Code Management system in conjunction with the GitHub online 
   // hosting system. The software in its entirety is available in the GitHub remote repository:
   // 
   //      https://github.com/practicalseries/PS2001-pal-software
   // 
   // The repository is public and can be freely copied (forked in GitHub terminology) and used 
   // under the MIT licence. 
   // 
   // The MIT licence is reproduced in full in the last network of this software module
   // 
   // 
   //  ———————————————————————————————————————————
   //  DATE     COMMIT TAG       AUTHOR        REASON FOR MODIFICATION
   //  ———————————————————————————————————————————
   //  2021.02.18    D0002      M. Gledhill      Baseline build
   // 
   //  2021.02.18    D0001      M. Gledhill      Hardware build
   // 
   //  2021.02.18    D0000      M. Gledhill      Initial commit — repository created
   //  ———————————————————————————————————————————
   // 
   // 
   // ▄▄▄▄▄▄▄▄▄▄▄▄▄▄▄▄▄▄▄▄▄▄▄▄▄▄▄▄▄▄▄▄▄▄▄▄▄▄▄▄▄▄▄▄
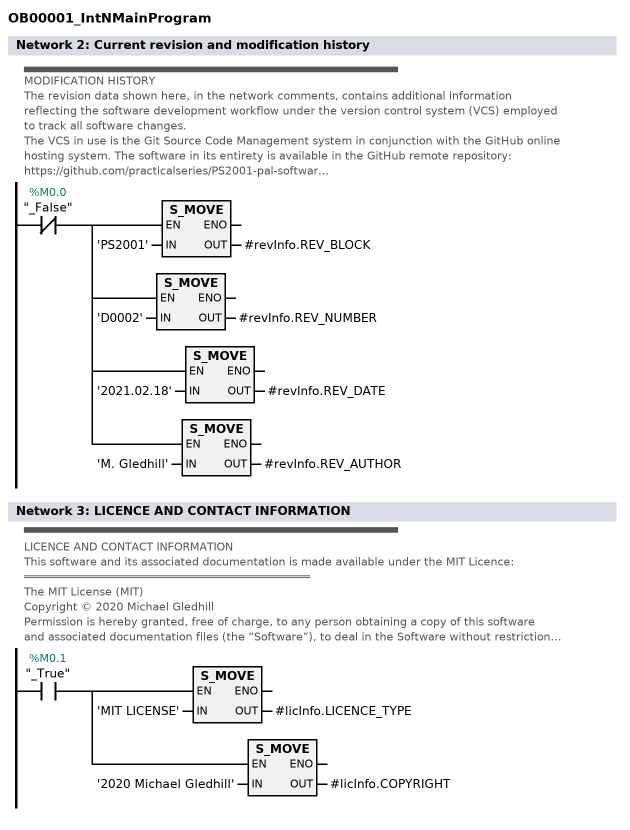
   RUNG wire#powerrail
      I_Contact( "_False" )
      wire#w1
      S_Move(in := 'PS2001', out => #revInfo.REV_BLOCK)
   END_RUNG
   RUNG wire#w1
      S_Move(in := 'D0002', out => #revInfo.REV_NUMBER)
   END_RUNG
   RUNG wire#w1
      S_Move(in := '2021.02.18', out => #revInfo.REV_DATE)
   END_RUNG
   RUNG wire#w1
      S_Move(in := 'M. Gledhill', out => #revInfo.REV_AUTHOR)
   END_RUNG
   // the same network as SCL:
   IF NOT "_False" THEN
       #revInfo.REV_BLOCK := 'PS2001';
       #revInfo.REV_NUMBER := 'D0002';
       #revInfo.REV_DATE := '2021.02.18';
       #revInfo.REV_AUTHOR := 'M. Gledhill';
   END_IF;
END_REGION

REGION Network 3: LICENCE AND CONTACT INFORMATION
   // ▀▀▀▀▀▀▀▀▀▀▀▀▀▀▀▀▀▀▀▀▀▀▀▀▀▀▀▀▀▀▀▀▀▀▀▀▀▀▀▀▀▀▀▀
   // LICENCE AND CONTACT INFORMATION
   // 
   // This software and its associated documentation is made available under the MIT Licence:
   // 
   // ════════════════════════════════════════════
   // 
   // The MIT License (MIT)
   // 
   // Copyright © 2020 Michael Gledhill
   // 
   // Permission is hereby granted, free of charge, to any person obtaining a copy of this software 
   // and associated documentation files (the “Software”), to deal in the Software without restriction, 
   // including without limitation the rights to use, copy, modify, merge, publish, distribute, 
   // sublicense, and/or sell copies of the Software, and to permit persons to whom the Software is 
   // furnished to do so, subject to the following conditions: 
   // 
   // The above copyright notice and this permission notice shall be included in all copies or 
   // substantial portions of the Software.
   // 
   // THE SOFTWARE IS PROVIDED “AS IS”, WITHOUT WARRANTY OF ANY KIND, EXPRESS OR IMPLIED, 
   // INCLUDING BUT NOT LIMITED TO THE WARRANTIES OF MERCHANTABILITY, FITNESS FOR A 
   // PARTICULAR PURPOSE AND NON-INFRINGEMENT. IN NO EVENT SHALL THE AUTHORS OR COPYRIGHT 
   // HOLDERS BE LIABLE FOR ANY CLAIM, DAMAGES OR OTHER LIABILITY, WHETHER IN AN ACTION OF 
   // CONTRACT, TORT OR OTHERWISE, ARISING FROM, OUT OF OR IN CONNECTION WITH THE SOFTWARE 
   // OR THE USE OR OTHER DEALINGS IN THE SOFTWARE.
   // 
   // ════════════════════════════════════════════
   //                    ┌────────────┐
   // You can reach the author by email here:   │  mg@practicalseries.com  │
   //                    └────────────┘
   // Questions, corrections, constructive criticism and complaints (polite ones) are invited.
   // 
   // ▄▄▄▄▄▄▄▄▄▄▄▄▄▄▄▄▄▄▄▄▄▄▄▄▄▄▄▄▄▄▄▄▄▄▄▄▄▄▄▄▄▄▄▄
   RUNG wire#powerrail
      Contact( "_True" )
      wire#w1
      S_Move(in := 'MIT LICENSE', out => #licInfo.LICENCE_TYPE)
   END_RUNG
   RUNG wire#w1
      S_Move(in := '2020 Michael Gledhill', out => #licInfo.COPYRIGHT)
   END_RUNG
   // the same network as SCL:
   IF "_True" THEN
       #licInfo.LICENCE_TYPE := 'MIT LICENSE';
       #licInfo.COPYRIGHT := '2020 Michael Gledhill';
   END_IF;
END_REGION
END_ORGANIZATION_BLOCK

FUNCTION "FC61000_DocGenExample" : Void   // FC61000, LAD
TITLE = Documentation - Gen — Example Documentation (full)
{ S7_Optimized_Access := 'TRUE' }
AUTHOR : M_Gledhill
FAMILY : Documentation
NAME : DocGenExample
VERSION : 1.0
// PRACTICAL SERIES AUTOMATION LIBRARY (PAL)   —   COPYRIGHT 2020 – M. GLEDHILL (MIT LICENCE)
//                   ———— ◆ ————
//  FOR DETAILED DOCUMENTATION — SELECT THE BLOCK IN THE PROJECT TREE AND PRESS SHIFT + F1
//  FULL ONLINE DOCUMENTATION IS AVAILABLE AT: https://practicalseries.com/2001-pal/index.html
// stored: AutoNumber false, IsIECCheckEnabled false, SetENOAutomatically false, UDAEnableTagReadback false
   VAR_TEMP
      revInfo : "UT01000_St_SysRevision";   // Revision information for this block
      licInfo : "UT01001_St_SysLicence";   // Licence information for this block
      wrkReal : Real;   // Working storage (real)
   END_VAR
   VAR CONSTANT
      _FALSE : Bool;   // Temporary internal "False" signal
   END_VAR
BEGIN

REGION Network 1: Block Contents
   // ▀▀▀▀▀▀▀▀▀▀▀▀▀▀▀▀▀▀▀▀▀▀▀▀▀▀▀▀▀▀▀▀▀▀▀▀▀▀▀▀▀▀▀▀
   // 
   // TITLE:    EXAMPLE DOCUMENTATION FOR USE IN COMMENTS
   // 
   // ▄▄▄▄▄▄▄▄▄▄▄▄▄▄▄▄▄▄▄▄▄▄▄▄▄▄▄▄▄▄▄▄▄▄▄▄▄▄▄▄▄▄▄▄
   // 
   // 
   // 
   // This block contains examples of all the typical forms of documentation used within the PAL
   // software. It provides the following:
   // 
   // CONTENTS (BY NETWORK)
   // 
   // NW 1.    Block Contents
   // NW 2.    Current revision and modification history
   // 
   // 
   // EXAMPLES
   // 
   // NW 3.    Example — Block description — Sections 1 to 3
   // NW 4.    Example — Block description — Sections 4 to 11
   // NW 5.    Example — Current revision and modification history
   // NW 6.    Example — Headings, lists and indented text
   // NW 7.    Example — Body text
   // NW 8.    Example — Standard Tables
   // NW 9.    Example — Other tables
   // NW 10.    Example — Equations
   // NW 11.    Example — Figures
   // 
   // 
   // CHARACTER LISTS
   // 
   // NW 12.    Special characters — Hyphens, whitespace and construction lines
   // NW 13.    Special characters — Arrows, box and block characters
   // NW 14.    Special characters — Currency, punctuation and full-width characters
   // NW 15.    Special characters — Greek, indexing characters and Roman numerals
   // NW 16.    Special characters — Mathematical operators (including vulgar fractions)
   // NW 17.    Special characters — Geometrical and ornamental characters
   // NW 18.    Special characters — Common character widths and additional whitespace characters
   // 
   // 
   // SPECIAL NETWORKS
   // 
   // NW 19.    OB1 NETWORK 1 — Project description
   // NW 20.    OB1 NETWORK 2 — Current revision and modification history
   // 
   // TYPICAL NETWORK COMMENTS
   // 
   // NW 21.    Load the system RTC and store in local variable  [typical network comment]
   // NW 22.    ██ STEP 03340 — DECLARATION (RUNNING)    [sequence network comment]
   // NW 23.       STEP 03340 — ACTION (INITIALISE)           [sequence network comment]
   // NW 24.       STEP 03340 — TRANSITION 01                   [sequence network comment]
   // NW 25.   LICENCE AND CONTACT INFORMATION       [final network]
   // 
   //               ━━━   ⬙⬙⬙⬙⬙⬙   ━━━
   // 
   // 
   // 
   // ▄▄▄▄▄▄▄▄▄▄▄▄▄▄▄▄▄▄▄▄▄▄▄▄▄▄▄▄▄▄▄▄▄▄▄▄▄▄▄▄▄▄▄▄
   // 1.     BLOCK TECHNICAL SUMMARY
   // 
   // 
   //  ――――――――――――――――――――――――――――――――――――――――――
   //  NOMENCLATURE & ADDRESSING
   //  ――――――――――――――――――――――――――――――――――――――――――
   //  BLOCK TITLE         Example Documentation for use in Comments
   //  BLOCK FUNCTION GROUP    Documentation
   //  BLOCK ADDRESS       FC 61000
   //  BLOCK SYMBOL        FC61000_DocGenExample
   //  BLOCK USER ID         DocGenExample
   // 
   //  ――――――――――――――――――――――――――――――――――――――――――
   //  BLOCK TYPE & USAGE
   //  ――――――――――――――――――――――――――――――――――――――――――
   //  BLOCK TYPE         Function (FC)
   //  BLOCK NUMBER        61000
   //  LANGUAGE           LAD
   //  OPTIMISED ACCESS     Yes
   //  PAL USAGE TYPE       Standard block
   // 
   //  ――――――――――――――――――――――――――――――――――――――――――
   //  METRICS
   //  ――――――――――――――――――――――――――――――――――――――――――
   //  EXECUTION TIME       24.48 μs¹
   //  LOAD MEMORY       50.26 kB  (51474 bytes)
   //  WORK MEMORY           0.34 kB      (347 bytes)
   //  ――――――――――――――――――――――――――――――――――――――――――
   //                ¹ Measured on: CPU-1515-2PN (order no. 6ES7 512-2AM02-0AB0)
   // 
   //                ━━━   ⬙⬙⬙⬙⬙⬙   ━━━
   // 
   // 
   // 
   // ▄▄▄▄▄▄▄▄▄▄▄▄▄▄▄▄▄▄▄▄▄▄▄▄▄▄▄▄▄▄▄▄▄▄▄▄▄▄▄▄▄▄▄▄
   // 2.     FUNCTIONAL DESCRIPTION
   // 
   // 
   // FC61000 is a documentation module that contains examples of all the common block and 
   // network comments used throughout the PAL software.
   // 
   // All examples are based upon the Style Guide (Doc. No. PS2001-5-2313-011).
   // 
   // FC61000 also contains lists of the characters available within the Siemens TIA font used within
   // all comment sections.
   // 
   //                ━━━   ⬙⬙⬙⬙⬙⬙   ━━━
   // 
   // 
   // 
   // ▄▄▄▄▄▄▄▄▄▄▄▄▄▄▄▄▄▄▄▄▄▄▄▄▄▄▄▄▄▄▄▄▄▄▄▄▄▄▄▄▄▄▄▄
   // 3.     DETAILED BLOCK DESCRIPTION
   // 
   // The purpose of this block is to provide an easy point of reference for the various documentation 
   // constructs and styles used within the PAL.
   // 
   // The block itself does not contain any executable code, with the exception of the revision and
   // licence networks, all networks are empty. The block itself does nothing, and its execution will
   // have no effect, other than extending the cycle time.
   // 
   //                ━━━   ⬙⬙⬙⬙⬙⬙   ━━━
   // 
   // 
   // 
   // ▄▄▄▄▄▄▄▄▄▄▄▄▄▄▄▄▄▄▄▄▄▄▄▄▄▄▄▄▄▄▄▄▄▄▄▄▄▄▄▄▄▄▄▄
   // 4.     PARAMETERS
   // 
   // 
   // This block has no parameters.
   // 
   //                ━━━   ⬙⬙⬙⬙⬙⬙   ━━━
   // 
   // 
   // 
   // ▄▄▄▄▄▄▄▄▄▄▄▄▄▄▄▄▄▄▄▄▄▄▄▄▄▄▄▄▄▄▄▄▄▄▄▄▄▄▄▄▄▄▄▄
   // 5.     DATA STRUCTURES AND USAGE (AND INSTANCE DATA BLOCKS)
   // 
   // 
   // The block has the following associated data structure:
   // 
   // 
   //  ――――――――――――――――――――――――――――――――――――――――――
   //  DATA STRUCTURE             DESCRIPTION
   //  ――――――――――――――――――――――――――――――――――――――――――
   //  UT01000_St_SysRevision          Revision information for this block    See FC01001
   //  UT01001_St_SysLicence           Licence information for this block  See FC01001
   //  ――――――――――――――――――――――――――――――――――――――――――
   // 
   //                ━━━   ⬙⬙⬙⬙⬙⬙   ━━━
   // 
   // 
   // 
   // ▄▄▄▄▄▄▄▄▄▄▄▄▄▄▄▄▄▄▄▄▄▄▄▄▄▄▄▄▄▄▄▄▄▄▄▄▄▄▄▄▄▄▄▄
   // 6.     CONSTANTS AND TEMPORARY (LOCAL) DATA
   // 
   // 
   // The following constants and temporary data storage are used:
   // 
   // 
   //  Temporary (local) data
   //  ――――――――――――――――――――――――――――――――――――――――――
   //  SIGNAL NAME          FUNCTION                  TYPE
   //  ――――――――――――――――――――――――――――――――――――――――――
   //  revInfo             Revision information for the block         UT01000
   //  licInfo           Licensing information for the block      UT01001
   //  wrkReal           Working storage (Real)             Real
   //  ――――――――――――――――――――――――――――――――――――――――――
   // 
   // 
   //  Constants data
   //  ――――――――――――――――――――――――――――――――――――――――――
   //  SIGNAL NAME          FUNCTION                  TYPE
   //  ――――――――――――――――――――――――――――――――――――――――――
   //  _FALSE            Temporary internal "False" signal      Bool
   //  ――――――――――――――――――――――――――――――――――――――――――
   // 
   // 
   //                ━━━   ⬙⬙⬙⬙⬙⬙   ━━━
   // 
   //  
   // 
   // ▄▄▄▄▄▄▄▄▄▄▄▄▄▄▄▄▄▄▄▄▄▄▄▄▄▄▄▄▄▄▄▄▄▄▄▄▄▄▄▄▄▄▄▄
   // 7.     BLOCK CALLS
   // 
   // 
   // There are no PAL block calls from within this block.
   // 
   //                ━━━   ⬙⬙⬙⬙⬙⬙   ━━━
   // 
   // 
   // 
   // ▄▄▄▄▄▄▄▄▄▄▄▄▄▄▄▄▄▄▄▄▄▄▄▄▄▄▄▄▄▄▄▄▄▄▄▄▄▄▄▄▄▄▄▄
   // 8.     ASSOCIATED BLOCKS
   // 
   // 
   // This is a stand-alone block and is not associated with any other blocks.
   // 
   //                ━━━   ⬙⬙⬙⬙⬙⬙   ━━━
   // 
   // 
   // 
   // 9.     SYSTEM BLOCK CALLS AND SYSTEM DATA TYPES
   // 
   // There are no system block calls.
   // 
   //                ━━━   ⬙⬙⬙⬙⬙⬙   ━━━
   // 
   // 
   // 
   // ▄▄▄▄▄▄▄▄▄▄▄▄▄▄▄▄▄▄▄▄▄▄▄▄▄▄▄▄▄▄▄▄▄▄▄▄▄▄▄▄▄▄▄▄
   // 10.     SPECIAL PROPERTIES AND REQUIREMENTS
   // 
   // 
   // 
   // ▂▂▂▂▂▂▂▂▂▂▂▂▂▂▂▂▂▂▂▂▂▂▂▂▂▂▂▂▂▂▂▂▂▂▂▂▂▂▂▂▂▂▂▂
   // 10.1   Block optimisation
   // 
   // 
   // Block optimisation is ACTIVE for this block
   // 
   // 
   // 
   // ▂▂▂▂▂▂▂▂▂▂▂▂▂▂▂▂▂▂▂▂▂▂▂▂▂▂▂▂▂▂▂▂▂▂▂▂▂▂▂▂▂▂▂▂
   // 10.2   Calling requirements
   // 
   // 
   // There are no special calling requirements for this block.
   // 
   //                ━━━   ⬙⬙⬙⬙⬙⬙   ━━━
   // 
   // 
   // 
   // ▄▄▄▄▄▄▄▄▄▄▄▄▄▄▄▄▄▄▄▄▄▄▄▄▄▄▄▄▄▄▄▄▄▄▄▄▄▄▄▄▄▄▄▄
   // 11.     EXAMPLE USAGE
   // 
   // 
   // The following shows a typical deployment of FC61000:
   // 
   // 
   //                       ┌────────────
   //    ───────────────────┤ FC61000 
   //                       ├──────────
   //                       │
   //                       │
   //                       │               │
   //                       │               │
   //                                    │
   //                       ─────────────┘
   // 
   //               ━━━   ⬙⬙⬙⬙⬙⬙   ━━━
   // 
   // 
   // ██████████████ █ █ █ █  END   █ █ █ █ ██████████████
END_REGION

REGION Network 2: Current revision and modification history
   // ▄▄▄▄▄▄▄▄▄▄▄▄▄▄▄▄▄▄▄▄▄▄▄▄▄▄▄▄▄▄▄▄▄▄▄▄▄▄▄▄▄▄▄▄
   // MODIFICATION HISTORY
   // 
   // The revision data shown here, in the network comments, contains additional information 
   // reflecting the software development workflow under the version control system (VCS) employed 
   // to track all software changes.
   // 
   // The VCS in use is the Git Source Code Management system in conjunction with the GitHub online 
   // hosting system. The software in its entirety is available in the GitHub remote repository:
   // 
   //      https://github.com/practicalseries/PS2001-pal-software
   // 
   // The repository is public and can be freely copied (forked in GitHub terminology) and used 
   // under the MIT licence. 
   // 
   // The MIT licence is reproduced in full in the last network of this software module
   // 
   // 
   //  ―――――――――――――――――――――――――――――――――――――――――――
   //  DATE       REVISION            MASTER BRANCH      DEV
   //          (nnn.amm)   COMMIT TAG    (Base ---> Merge)    BRANCH   Author
   //  ———————————————————————————————————————————
   //  2021.02.18    001.000   D0002      D0001 D0002  None    M. Gledhill
   //                        FC61000 — RELEASED FOR USE
   //                          Block imported form 000.125-Db
   //  ———————————————————————————————————————————
   //   Where: nnn  =  Major revision
   //         a  =  Type (1-7 Development, 8 Proving, 9 Qualification, 0 Release)
   //       mm  =  Minor revision (must be 00 if a = 0)
   //         Block properties version number should be set to nn.a (only one decimal place)
   // 
   // ▄▄▄▄▄▄▄▄▄▄▄▄▄▄▄▄▄▄▄▄▄▄▄▄▄▄▄▄▄▄▄▄▄▄▄▄▄▄▄▄▄▄▄▄
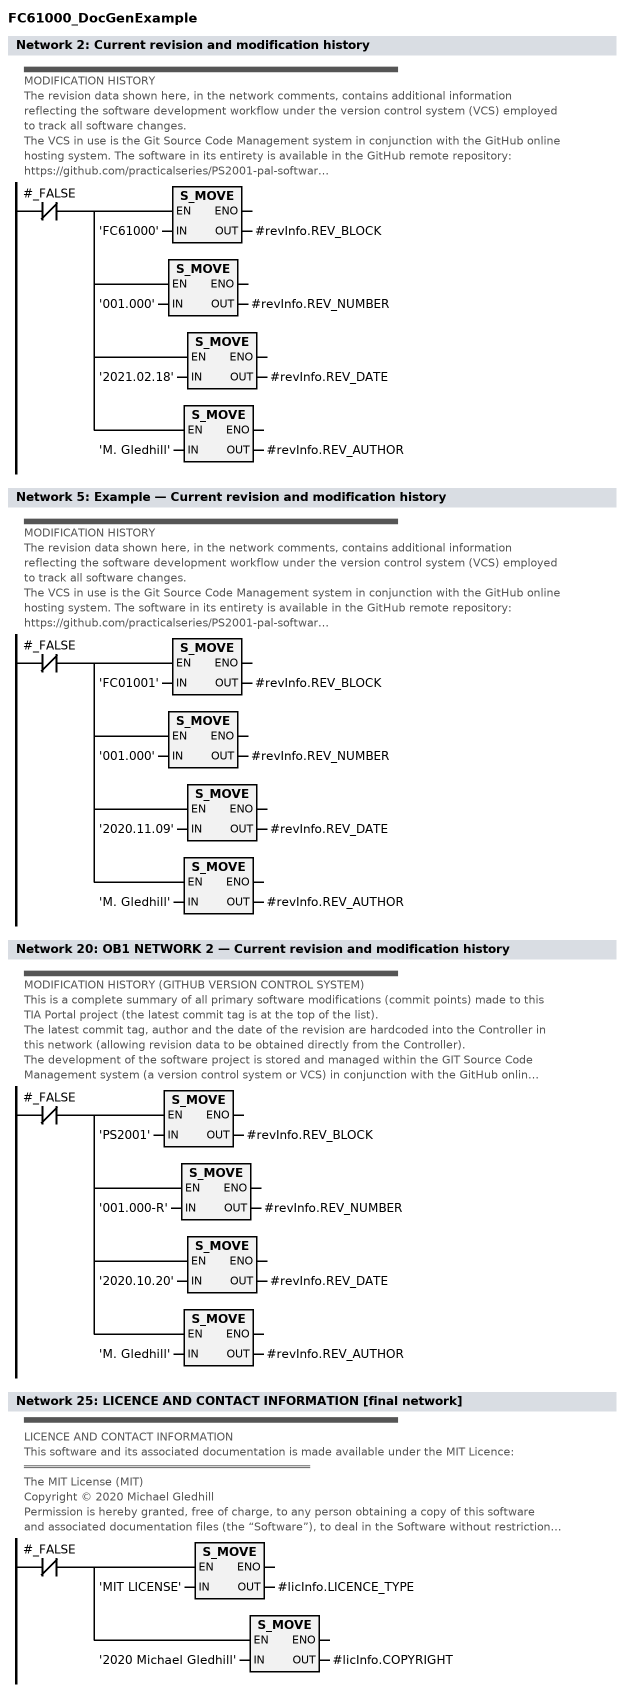
   RUNG wire#powerrail
      I_Contact( #_FALSE )
      wire#w1
      S_Move(in := 'FC61000', out => #revInfo.REV_BLOCK)
   END_RUNG
   RUNG wire#w1
      S_Move(in := '001.000', out => #revInfo.REV_NUMBER)
   END_RUNG
   RUNG wire#w1
      S_Move(in := '2021.02.18', out => #revInfo.REV_DATE)
   END_RUNG
   RUNG wire#w1
      S_Move(in := 'M. Gledhill', out => #revInfo.REV_AUTHOR)
   END_RUNG
   // the same network as SCL:
   IF NOT #_FALSE THEN
       #revInfo.REV_BLOCK := 'FC61000';
       #revInfo.REV_NUMBER := '001.000';
       #revInfo.REV_DATE := '2021.02.18';
       #revInfo.REV_AUTHOR := 'M. Gledhill';
   END_IF;
END_REGION

REGION Network 3: Example — Block description — Sections 1 to 3
   // | ▀▀▀▀▀▀▀▀▀▀▀▀▀▀▀▀▀▀▀▀▀▀▀▀▀▀▀▀▀▀▀▀▀▀▀▀▀▀▀▀▀▀▀▀
   // 
   // TITLE:    SUBROUTINE — EVENT TIMER USING RTC
   // 
   // ▄▄▄▄▄▄▄▄▄▄▄▄▄▄▄▄▄▄▄▄▄▄▄▄▄▄▄▄▄▄▄▄▄▄▄▄▄▄▄▄▄▄▄▄
   //  
   // 
   // 
   // This block (FC18151_SubTimeEventRTC) is a subroutine block that times the duration of an event 
   // to nanosecond resolution.
   // 
   // The block records the time the event started (rising edge of the TRIGGER signal), the time the 
   // event ended (falling edge of the TRIGGER signal) and calculates the duration of the event (end 
   // time minus the start time).
   // 
   // The start and end times are read from the real time clock of the controller.
   // 
   // This is a subroutine block.
   // 
   // 
   // 
   // ▄▄▄▄▄▄▄▄▄▄▄▄▄▄▄▄▄▄▄▄▄▄▄▄▄▄▄▄▄▄▄▄▄▄▄▄▄▄▄▄▄▄▄▄
   // 1.     BLOCK TECHNICAL SUMMARY
   // 
   // 
   //  ――――――――――――――――――――――――――――――――――――――――――
   //  NOMENCLATURE & ADDRESSING
   //  ――――――――――――――――――――――――――――――――――――――――――
   //  BLOCK TITLE         Subroutine Event Timer using RTC
   //  BLOCK FUNCTION GROUP    Subroutine
   //  BLOCK ADDRESS       FC18151
   //  BLOCK SYMBOL        FC18151_SubTimeEventRTC
   //  BLOCK USER ID         SubTimeEventRTC
   // 
   //  ――――――――――――――――――――――――――――――――――――――――――
   //  BLOCK TYPE & USAGE
   //  ――――――――――――――――――――――――――――――――――――――――――
   //  BLOCK TYPE         Function (FC)
   //  BLOCK NUMBER        18151
   //  LANGUAGE           LAD
   //  OPTIMISED ACCESS     Yes
   //  PAL USAGE TYPE       Standard block
   // 
   //  ――――――――――――――――――――――――――――――――――――――――――
   //  METRICS
   //  ――――――――――――――――――――――――――――――――――――――――――
   //  EXECUTION TIME       18.41 μs¹
   //  LOAD MEMORY       23.11 kB  (23667 bytes)
   //  WORK MEMORY           0.43 kB      (442 bytes)
   //  ――――――――――――――――――――――――――――――――――――――――――
   //                ¹ Measured on: CPU-1515-2PN (order no. 6ES7 512-2AM02-0AB0)
   // 
   // 
   // ▄▄▄▄▄▄▄▄▄▄▄▄▄▄▄▄▄▄▄▄▄▄▄▄▄▄▄▄▄▄▄▄▄▄▄▄▄▄▄▄▄▄▄▄
   // 2.     FUNCTIONAL DESCRIPTION
   // 
   // 
   // FC18151 is the Subroutine Event Timer using RTC block, it simply records the duration of an event 
   // with a high degree of accuracy. The event being timed is a Boolean signal passed to the block as 
   // the TRIGGER parameter.
   // 
   // Three times are recorded for the event, the start time (rising edge of the TRIGGER parameter), the 
   // end time (falling edge of the TRIGGER parameter) and the duration of the event (end time minus 
   // the start time). The duration is calculated on the falling edge of the TRIGGER parameter, 
   // immediately after the end time is recorded.
   // 
   // The start and end times are read from the Controller’s internal real time clock (RTC) and are 
   // stored in DTL (date time long) format, this format contains year, month, day, hours, minutes, 
   // seconds, milliseconds, microseconds and nano seconds.
   // 
   // The duration is stored in LTime (long time, 64-bit) format, and is very accurate, it resolves to 
   // days, hours, minutes, seconds milliseconds, microseconds and nanoseconds, it keeps this 
   // resolution irrespective of the duration.
   // 
   // The duration is also calculated as a real number in seconds (or fractions thereof); this is a 
   // more convenient format for holding the duration, but is not as accurate as the LTime format.
   // 
   // 
   // 
   // 
   // 
   // ▄▄▄▄▄▄▄▄▄▄▄▄▄▄▄▄▄▄▄▄▄▄▄▄▄▄▄▄▄▄▄▄▄▄▄▄▄▄▄▄▄▄▄▄
   // 3.     DETAILED BLOCK DESCRIPTION
   // 
   // The purpose of this block is to determine with a high degree of accuracy the duration of an event, 
   // the event itself must be in the form of a Boolean trigger signal, the rising edge of the signal is 
   // considered to be the start of the event and the falling edge the end of the event.
   // 
   // The event signal is passed to the block as the TRIGGER parameter. 
   // The block returns five values, these are stored in a UDT passed to the block in the 
   // DYNAMIC_DATA parameter: 
   // 
   //  ――――――――――――――――――――――――――――――――――――――――――
   //  PARAM         ASSOCIATED UDT            ASSOCIATED DATA BLOCK
   //  ――――――――――――――――――――――――――――――――――――――――――
   //  DYNAMIC_DATA     UT38151_Dy_SubTimeEventRTC       DB38151_Dy_SubTimeEventRTC
   //  ――――――――――――――――――――――――――――――――――――――――――
   // 
   // 
   // The block returns the following data:
   // 
   //  UT38151_Dy_SubTimeEventRTC
   //  ―――――――――――――――――――――――――――――――――――――――――― 
   //  SIGNAL NAME          FUNCTION                     TYPE
   //  ――――――――――――――――――――――――――――――――――――――――――
   //  status_Running      STATUS — The event timer is running         Bool
   // 
   //  actual_StartTime      ACTUAL — Time at which the TRIGGER signal        DTL
   //                      went high (event start time)
   // 
   //  actual_EndTime        ACTUAL — Time at which the TRIGGER signal     DTL
   //                      went low (event end time)
   // 
   //  actual_Duration        ACTUAL — Event duration              LTime
   // 
   //  actual_DurationSec       ACTUAL — Event duration in seconds           REAL
   //  ――――――――――――――――――――――――――――――――――――――――――
   //  Block returned signals
   // 
   // 
   // 
   // ▂▂▂▂▂▂▂▂▂▂▂▂▂▂▂▂▂▂▂▂▂▂▂▂▂▂▂▂▂▂▂▂▂▂▂▂▂▂▂▂▂▂▂▂
   // 3.1     Timing an event
   // 
   // The block constantly monitors the TRIGGER parameter; if a rising edge is seen on the TRIGGER 
   // parameter (point ① in the figure below), the Controller RTC is read and its value is stored in 
   // actual_StartTime, at the same time the running signal (status_Running) is activated.
   // 
   // The block continues to monitor the TRIGGER parameter, when a falling edge is detected 
   // (point ②), the RTC is read once more and its value is stored in actual_EndTime, and the running 
   // signal (status_Running) is deactivated.
   // 
   // Once the end time is stored, the following calculation is carried out:
   // 
   // 
   // ┌───────────────────────────┐
   // │ actual_Duration =  actual_EndTime ─ actual_StartTime    │
   // └───────────────────────────┘
   // 
   // 
   //                     ①            ②
   //   TRIGGER │             ┏━━━━━━━━━━━━┓
   //         │             ┃               ┃
   //         │             ┃               ┃
   //         │             ┃               ┃
   //         │             ┃               ┃                              
   //         ┼━━━━━━━━━━━━╶╶╶╶╶╶╶╶╶╶╶╶╶━━━━━━━━━━ time
   //                  ↗             ↖
   //            actual_StartTime ╎            ╎ actual_EndTime
   //    DTL#2020-04-18-09:34:25.899548353        DTL#2020-04-18-09:34:36.004744916
   // 
   //                    ╎               ╎                      actual_Duration
   //                                      LT#10S_105MS_196US_563NS
   //                    ╎               ╎  
   //                                                     actual_DurationSec
   //                    ╎               ╎                              10.10519
   // 
   //         │status_Running      ┏━━━━━━━━━━━━┓
   //         │             ┃               ┃
   //         │             ┃               ┃
   //         │             ┃               ┃
   //         │             ┃               ┃
   //         ┼━━━━━━━━━━━━╶╶╶╶╶╶╶╶╶╶╶╶╶━━━━━━━━━━
   // 
   // 
   // 
   // ▂▂▂▂▂▂▂▂▂▂▂▂▂▂▂▂▂▂▂▂▂▂▂▂▂▂▂▂▂▂▂▂▂▂▂▂▂▂▂▂▂▂▂▂
   // 3.1     Date and time data types
   // 
   // Both the start and end times (actual_StartTime and actual_EndTime) are of the type DTL 
   // (date time long), this itself is a data structure in the form:
   // 
   //  DTL Data Structure
   //  ――――――――――――――――――――――――――――――――――――――――――
   //  SIGNAL NAME          FUNCTION                     TYPE
   //  ――――――――――――――――――――――――――――――――――――――――――
   //  YEAR             Year (returns a value in the range 1970 to 2262)     UInt
   //  MONTH            Month (1-12 representing Jan to Dec)        USInt
   //  DAY              Day of month (1-31)                USInt
   //  WEEKDAY          Day of week (1-7, where 1=Sunday, 7=Saturday)    USInt
   //  HOUR           Hour of day (0-23)                   USInt
   //  MINUTE           Minutes (0-59)                   USInt
   //  SECOND            Seconds (0-59)                  USInt
   //  NANOSECOND        Nanoseconds (0-999,999,999)           UDint
   //  ――――――――――――――――――――――――――――――――――――――――――
   // 
   // When displayed, it has the format:
   // 
   //       DTL#2020-04-18-09:34:25.899548353
   // 
   //  I.e.      18th April 2020 at 09:43:25 AM and 899,548,353 ns.
   // 
   // The calculated duration (actual_Duration) is of data type LTime (long time).
   // 
   // The LTime data type is essentially an 8-byte number (64-bit number) that stores a time value in 
   // nanoseconds. In the above example, the actual_Duration has the formatted value of:
   // 
   //       LT#10S_105MS_196US_563NS
   // 
   //  I.e.      10 seconds, 105 milliseconds, 196 microseconds and 563 nanoseconds.
   // 
   // It is shown in this format, because TIA portal understands the LTime data type and is able to 
   // interpret the value as days, hours, minute, seconds, milliseconds, microseconds and 
   // nanoseconds. 
   // 
   // In practice, the actual_Duration simply (in this example) holds a very large number:
   // 
   //       10,105,196,563
   // 
   // This is the duration of the event in nanoseconds (i.e. 10,105,196,563 nanoseconds). To convert 
   // the number to seconds, simply divide by 1,000,000,000 (or 1 × 10^9); this would give:
   // 
   //       10.105196563 seconds
   // 
   // The reason the duration is specified as an LTime rather that DTL is that, somewhat confusingly, 
   // DTL is a relative measure of time (relative to 1st January, 1970), if the above duration were 
   // represented as a DTL value it would read:
   // 
   //       DTL#1970-01-01-00:00:10.105196563
   // 
   // Hours, minutes and seconds are OK, but the date part doesn’t make sense (to make it 
   // meaningful, 1970 must be subtracted from the YEAR value and 1 from both the MONTH and 
   // DAY values).
   // 
   // The LTime data type can store a duration of up to 106,751 days (about 300 years) and while not 
   // perfect, it seems long enough for most practical situations (possibly not for geological 
   // applications).
   // 
   // The actual_Duration in LTime format is very accurate, but it is an unwieldly data type, to provide a 
   // more user friendly (although less accurate) format, the actual_Duration signal is converted to a 
   // real number giving the duration in seconds, this is stored in the actual_DurationSec signal. In the 
   // above example: 
   // 
   //       actual_DurationSec has the value 10.10519 seconds
   // 
   // It is less accurate, it does not resolve to nanoseconds; however, it is easier to use and display 
   // and is accurate enough for most applications.
   // 
   // 
   // 
   // ▁▁▁▁▁▁▁▁▁▁▁▁▁▁▁▁▁▁▁▁▁▁▁▁▁▁▁▁▁▁▁▁▁▁▁▁▁▁▁▁▁▁▁▁
   // A note on real numbers
   // 
   // The LTime format is very accurate, it is basically counting nanoseconds, and because it is 64-bits 
   // long it can count up to very high values (about 584 years at nanosecond resolution).
   // 
   // Real numbers however, are limited to 32-bits and suffer from precision loss, this results from the 
   // fact that the real number has an accuracy of “about” 7 decimal digits, for example 20365.45, 
   // 20.43728, 1.482967, 0.3356428, &c. Essentially, the bigger the number, the fewer the decimal 
   // places — a total of 7 decimal digits.
   // 
   // Very big and very small numbers can be represented by adding trailing zeros for big numbers 
   // (e.g. 3275625000) and leading zeros for small numbers (0.000003275625) in both these 
   // examples, there are only 7 decimal digits, just shifted effectively left or right.
   // 
   // This type of representation is usually handled by applying scientific notation, the number 
   // 1,568,497,000,000 would be represented as 1.568497 × 10^12, it only has 7 decimal digits, 
   // the number 1,568,497,132,792, would be represented as exactly the same value, the 132,792 
   // part of the number cannot be resolved and are lost.
   // 
   // 
   // 
   // 
   //                ━━━   ⬙⬙⬙⬙⬙⬙   ━━━
END_REGION

REGION Network 4: Example — Block description — Sections 4 to 11
   // ▄▄▄▄▄▄▄▄▄▄▄▄▄▄▄▄▄▄▄▄▄▄▄▄▄▄▄▄▄▄▄▄▄▄▄▄▄▄▄▄▄▄▄▄
   // 4.     PARAMETERS
   // 
   // 
   // The following parameters are associated with the block:
   // 
   //  
   //  ――――――――――――――――――――――――――――――――――――――――――
   //  PARAM         FUNCTION                    TYPE      IN-OUT 
   //  ――――――――――――――――――――――――――――――――――――――――――
   //  SYS_SIGNALS      Common system signals              UT21000    In
   //           logic and timing signals for parametric access
   // 
   //  TRIGGER       Event trigger signal (a rising edge marks the     Bool   In
   //           start of the event, the falling edge the end)
   // 
   //  STATIC_DATA     Data structure that holds the configuration data     UT02001    In
   // 
   //  DYNAMIC_DATA      Stores the results of the event timing       UT38151    InOut
   //  ――――――――――――――――――――――――――――――――――――――――――
   // 
   //                ━━━   ⬙⬙⬙⬙⬙⬙   ━━━
   // 
   // 
   // 
   // ▄▄▄▄▄▄▄▄▄▄▄▄▄▄▄▄▄▄▄▄▄▄▄▄▄▄▄▄▄▄▄▄▄▄▄▄▄▄▄▄▄▄▄▄
   // 5.     DATA STRUCTURES AND USAGE (AND INSTANCE DATA BLOCKS)
   // 
   // 
   // The block has the following associated data structure:
   // 
   // 
   //  ――――――――――――――――――――――――――――――――――――――――――
   //  DATA STRUCTURE             DESCRIPTION
   //  ――――――――――――――――――――――――――――――――――――――――――
   //  UT01000_St_SysRevision          Revision information for this block    See FC01001
   //  UT01001_St_SysLicence           Licence information for this block  See FC01001
   //  UT21000_Dy_SysSignals           System signals for logic and timing  See FC01001
   //  UT38151_Dy_SubTimeEventRTC        Dynamic data structure for the event timing block
   //  ――――――――――――――――――――――――――――――――――――――――――
   // 
   // 
   // 
   // ▂▂▂▂▂▂▂▂▂▂▂▂▂▂▂▂▂▂▂▂▂▂▂▂▂▂▂▂▂▂▂▂▂▂▂▂▂▂▂▂▂▂▂▂
   // 5.1     UT38151_Dy_TimeEventRTC
   // 
   // Stores the timing values for the event:
   // 
   //  UT38151_Dy_TimeEventRTC
   //  ――――――――――――――――――――――――――――――――――――――――――
   //  SIGNAL NAME          FUNCTION                     TYPE
   //  ――――――――――――――――――――――――――――――――――――――――――
   //  status_Running      STATUS — The event timer is running         Bool
   // 
   //  actual_StartTime      ACTUAL — Time at which the TRIGGER signal        DTL
   //                      went high (event start time)
   // 
   //  actual_EndTime        ACTUAL — Time at which the TRIGGER signal     DTL
   //                      went low (event end time)
   // 
   //  actual_Duration        ACTUAL — Event duration              LTime
   // 
   //  actual_DurationSec       ACTUAL — Event duration in seconds           REAL
   //  ――――――――――――――――――――――――――――――――――――――――――
   // 
   //                ━━━   ⬙⬙⬙⬙⬙⬙   ━━━
   // 
   // 
   // 
   // ▄▄▄▄▄▄▄▄▄▄▄▄▄▄▄▄▄▄▄▄▄▄▄▄▄▄▄▄▄▄▄▄▄▄▄▄▄▄▄▄▄▄▄▄
   // 6.     CONSTANTS AND TEMPORARY (LOCAL) DATA
   // 
   // 
   // The following constants and temporary data storage are used:
   // 
   // 
   //  Temporary (local) data
   //  ――――――――――――――――――――――――――――――――――――――――――
   //  SIGNAL NAME          FUNCTION                  TYPE
   //  ――――――――――――――――――――――――――――――――――――――――――
   //  revInfo             Revision information for the block         UT01000
   //  licInfo           Licensing information for the block      UT01001
   //  wrkInt           Working storage area (integer)          Int
   //  wrkReal           Working storage (Real)             Real
   //  wrkLInt            Working storage area (long integer)        LInt
   //  ――――――――――――――――――――――――――――――――――――――――――
   // 
   //                ━━━   ⬙⬙⬙⬙⬙⬙   ━━━
   // 
   // 
   // 
   // ▄▄▄▄▄▄▄▄▄▄▄▄▄▄▄▄▄▄▄▄▄▄▄▄▄▄▄▄▄▄▄▄▄▄▄▄▄▄▄▄▄▄▄▄
   // 7.     BLOCK CALLS
   // 
   // 
   // There are no PAL block calls from within this block.
   // 
   //                ━━━   ⬙⬙⬙⬙⬙⬙   ━━━
   // 
   // 
   // 
   // ▄▄▄▄▄▄▄▄▄▄▄▄▄▄▄▄▄▄▄▄▄▄▄▄▄▄▄▄▄▄▄▄▄▄▄▄▄▄▄▄▄▄▄▄
   // 8.     ASSOCIATED BLOCKS
   // 
   // 
   // This is a stand-alone block and is not associated with any other blocks.
   // 
   //                ━━━   ⬙⬙⬙⬙⬙⬙   ━━━
   // 
   // 
   // 
   // ▄▄▄▄▄▄▄▄▄▄▄▄▄▄▄▄▄▄▄▄▄▄▄▄▄▄▄▄▄▄▄▄▄▄▄▄▄▄▄▄▄▄▄▄
   // 9.     SYSTEM BLOCK CALLS AND SYSTEM DATA TYPES
   // 
   // 
   // The following calls are made to system blocks:
   // 
   // 
   //  System block calls
   //  ――――――――――――――――――――――――――――――――――――――――――
   //  BLOCK          TITLE             DESCRIPTION  
   //  ――――――――――――――――――――――――――――――――――――――――――
   //  RD_LOC_T             Read the local RTC time    Reads the CPU real time clock 
   //  ――――――――――――――――――――――――――――――――――――――――――
   // 
   // There are no special system data types used.
   // 
   // 
   //                ━━━   ⬙⬙⬙⬙⬙⬙   ━━━
   // 
   // 
   // 
   // ▄▄▄▄▄▄▄▄▄▄▄▄▄▄▄▄▄▄▄▄▄▄▄▄▄▄▄▄▄▄▄▄▄▄▄▄▄▄▄▄▄▄▄▄
   // 10.     SPECIAL PROPERTIES AND REQUIREMENTS
   // 
   // 
   // 
   // ▂▂▂▂▂▂▂▂▂▂▂▂▂▂▂▂▂▂▂▂▂▂▂▂▂▂▂▂▂▂▂▂▂▂▂▂▂▂▂▂▂▂▂▂
   // 10.1   Block optimisation
   // 
   // 
   // Block optimisation is ACTIVE for this block
   // 
   // 
   // 
   // ▂▂▂▂▂▂▂▂▂▂▂▂▂▂▂▂▂▂▂▂▂▂▂▂▂▂▂▂▂▂▂▂▂▂▂▂▂▂▂▂▂▂▂▂
   // 10.2   Calling requirements
   // 
   // 
   // There are no special calling requirements for this block.
   // 
   // 
   // 
   // ▂▂▂▂▂▂▂▂▂▂▂▂▂▂▂▂▂▂▂▂▂▂▂▂▂▂▂▂▂▂▂▂▂▂▂▂▂▂▂▂▂▂▂▂
   // 10.3   Other properties
   // 
   // 
   // This block does not require the usual SYS_SIGNALS logic and timing data.
   // 
   // 
   //                ━━━   ⬙⬙⬙⬙⬙⬙   ━━━
   // 
   // 
   // 
   // ▄▄▄▄▄▄▄▄▄▄▄▄▄▄▄▄▄▄▄▄▄▄▄▄▄▄▄▄▄▄▄▄▄▄▄▄▄▄▄▄▄▄▄▄
   // 11.     EXAMPLE USAGE
   // 
   // 
   // The following shows a typical deployment of FC18151:
   // 
   //                      ┌─────────────
   //        ──────────────┤ FC18151
   //                      ├───────────
   //                 %M100.0    │
   //               "Event001"   ─┤ TRIGGER
   //                      │
   //     "DB38151_Dy_TimeEventRTC".Event001 ─┤ DYNAMIC_DATA
   //                      │
   //                      │             │
   //                                    │
   //                           ─────────┘
   // 
   //               ━━━   ⬙⬙⬙⬙⬙⬙   ━━━
   // 
   // 
   // ██████████████ █ █ █ █  END   █ █ █ █ ██████████████
END_REGION

REGION Network 5: Example — Current revision and modification history
   // ▄▄▄▄▄▄▄▄▄▄▄▄▄▄▄▄▄▄▄▄▄▄▄▄▄▄▄▄▄▄▄▄▄▄▄▄▄▄▄▄▄▄▄▄
   // MODIFICATION HISTORY
   // 
   // 
   // The revision data shown here, in the network comments, contains additional information 
   // reflecting the software development workflow under the version control system (VCS) employed 
   // to track all software changes.
   // 
   // The VCS in use is the Git Source Code Management system in conjunction with the GitHub online 
   // hosting system. The software in its entirety is available in the GitHub remote repository:
   // 
   //      https://github.com/practicalseries/PS2001-pal-software
   // 
   // The repository is public and can be freely copied (forked in GitHub terminology) and used 
   // under the MIT licence. 
   // 
   // The MIT licence is reproduced in full in the last network of this software module
   // 
   // 
   //  ―――――――――――――――――――――――――――――――――――――――――――
   //  DATE       REVISION            MASTER BRANCH      DEV
   //          (nnn.amm)   COMMIT TAG    (Base ---> Merge)    BRANCH   Author
   //  ———————————————————————————————————————————
   //  2020.11.09    001.000   D0003      D0002 D0003  None    M. Gledhill
   //                        FC01001 — RELEASED FOR USE
   //                          Merge back to master branch
   //  
   //  2020.11.09    001.000   D0002A-001.000  D0002 N/A     D0002A   M. Gledhill
   //                        FC01001 — Post test released for use
   // 
   //  2020.11.08    000.801   D0002A-000.801  D0002 N/A     D0002A   M. Gledhill
   //                        FC01001 — Released for SMT
   // 
   //  2020.11.04    000.102   D0002A-000.102  D0002 N/A     D0002A   M. Gledhill
   //                        FC01001 — Incremental build
   // 
   //  2020.11.03    000.101   D0002A-000.101  D0002 N/A     D0002A   M. Gledhill
   //                        FC01001 — Block created
   //  ———————————————————————————————————————————
   //   Where: nnn  =  Major revision
   //         a  =  Type (1-7 Development, 8 Proving, 9 Qualification, 0 Release)
   //       mm  =  Minor revision (must be 00 if a = 0)
   //         Block properties version number should be set to nn.a (only one decimal place)
   // 
   // ▄▄▄▄▄▄▄▄▄▄▄▄▄▄▄▄▄▄▄▄▄▄▄▄▄▄▄▄▄▄▄▄▄▄▄▄▄▄▄▄▄▄▄▄
   RUNG wire#powerrail
      I_Contact( #_FALSE )
      wire#w1
      S_Move(in := 'FC01001', out => #revInfo.REV_BLOCK)
   END_RUNG
   RUNG wire#w1
      S_Move(in := '001.000', out => #revInfo.REV_NUMBER)
   END_RUNG
   RUNG wire#w1
      S_Move(in := '2020.11.09', out => #revInfo.REV_DATE)
   END_RUNG
   RUNG wire#w1
      S_Move(in := 'M. Gledhill', out => #revInfo.REV_AUTHOR)
   END_RUNG
   // the same network as SCL:
   IF NOT #_FALSE THEN
       #revInfo.REV_BLOCK := 'FC01001';
       #revInfo.REV_NUMBER := '001.000';
       #revInfo.REV_DATE := '2020.11.09';
       #revInfo.REV_AUTHOR := 'M. Gledhill';
   END_IF;
END_REGION

REGION Network 6: Example — Headings, lists and indented text
   // ▀▀▀▀▀▀▀▀▀▀▀▀▀▀▀▀▀▀▀▀▀▀▀▀▀▀▀▀▀▀▀▀▀▀▀▀▀▀▀▀▀▀▀▀
   // 
   // TITLE:    HEADINGS, LISTS AND INDENTED TEXT
   // 
   // ▄▄▄▄▄▄▄▄▄▄▄▄▄▄▄▄▄▄▄▄▄▄▄▄▄▄▄▄▄▄▄▄▄▄▄▄▄▄▄▄▄▄▄▄
   // 
   //                ━━━   ⬙⬙⬙⬙⬙⬙   ━━━[1 empty line above, 3 empty lines below]
   // 
   // 
   // 
   // ▄▄▄▄▄▄▄▄▄▄▄▄▄▄▄▄▄▄▄▄▄▄▄▄▄▄▄▄▄▄▄▄▄▄▄▄▄▄▄▄▄▄▄▄[3 empty lines above, 5 if no ⬙ flourish]
   // 1.     [MAIN SECTION — ALL UPPERCASE — IF UNNUMBERED STARTS AT LEFT EDGE]
   // 10.     [MAIN SECTION — ALL UPPERCASE — IF UNNUMBERED STARTS AT LEFT EDGE]
   // 
   // 
   // 
   // ▂▂▂▂▂▂▂▂▂▂▂▂▂▂▂▂▂▂▂▂▂▂▂▂▂▂▂▂▂▂▂▂▂▂▂▂▂▂▂▂▂▂▂▂[3 empty lines above]
   // 1.1     [Subsection, two single digits   — Sentence case — if unnumbered, starts at left edge]
   // 10.1   [Subsection, one double digit   — Sentence case — if unnumbered, starts at left edge]
   // 10.10    [Subsection, two double digits — Sentence case — if unnumbered, starts at left edge]
   // 
   // 
   // 
   // ▁▁▁▁▁▁▁▁▁▁▁▁▁▁▁▁▁▁▁▁▁▁▁▁▁▁▁▁▁▁▁▁▁▁▁▁▁▁▁▁▁▁▁▁[3 empty lines above]
   // 1.1.1     [Inline, three single digits   — Sentence case — if unnumbered, starts at left edge]
   // 10.1.1   [Inline, one double digit   — Sentence case — if unnumbered, starts at left edge]
   // 10.10.1   [Inline, two double digits    — Sentence case — if unnumbered, starts at left edge]
   // 10.10.10 [Inline, three double digits — Sentence case — if unnumbered, starts at left edge]
   // 
   // 
   //    •   [Lists — non-numbered]
   //    ① [Lists — numbered]
   //    1.  [Lists — numbered single digit   — less than 10 entries]
   //      1.  [Lists — numbered single digit   — 10 or more entries]
   //    10.  [Lists — numbered double digit — 10 or more entries]
   // 
   //    1.  Communication handling
   //      Executes system to system communications (Controller to Controller, point-to-point,
   //      ProfiBus FMS &c.)
   //    2.  Subroutine functions
   //      Various subroutines (called by other block) to execute particular functions 
   //      (subroutines are organised into similar function areas)
   //    3.  Normal (non-error) interrupt functions
   //      Usually associated with specific OBs, interrupts generated by standard system events
   //      (time of day, cyclic, hardware &c.)
   // 
   // Note:    Bipolar and unipolar instruments have different tolerances, a 0-20 mA unipolar signal
   //      has a full instrument range of 16 mA and the 2.5% tolerance will thus be ±0.4 mA 
   // 
   // ――――――――――
   // ¹         Footnotes can use the characters ¹, ² and ³ to indicate the footnote number
   //      Second lines are identical to those for notes.
   // ――――――――――
   // 
   // 
   //                ━━━   ⬙⬙⬙⬙⬙⬙   ━━━
   // 
   // 
   // ██████████████ █ █ █ █  END   █ █ █ █ ██████████████
END_REGION

REGION Network 7: Example — Body text
   // ▀▀▀▀▀▀▀▀▀▀▀▀▀▀▀▀▀▀▀▀▀▀▀▀▀▀▀▀▀▀▀▀▀▀▀▀▀▀▀▀▀▀▀▀
   // 
   // TITLE:    BODY TEXT (AN EXAMPLE)
   // 
   // ▄▄▄▄▄▄▄▄▄▄▄▄▄▄▄▄▄▄▄▄▄▄▄▄▄▄▄▄▄▄▄▄▄▄▄▄▄▄▄▄▄▄▄▄
   // 
   // 
   // 
   // Normal (body) text is left justified to the left hand edge of the comment area; manual line-breaks
   // must be inserted when the text exceeds the range of the title bars (lines at the top of this block
   // and above each section and subsection — exactly 44 em-spaces).
   // 
   // The following fragment highlights this: 
   // 
   // The alignments in Figure 7.4 are such that the leading edge (left side) of any indented character
   // is aligned with the leading edge of an em-space in a line of em-spaces that span the page (this
   // can be seen with the chequered patterns in the screen shot — all indents line up with the left
   // edge of an em-space).
   // 
   // The problem with this is that the alphanumeric characters are not all the same width and
   // generally, they are not one em-space wide (there are no characters that are one em wide, not
   // even the M, which is odd given that that is how the em unit was derived, see here).
   // With the TIA Portal font, one em is exactly the same width as four normal space characters (a 
   // normal space being the character entered when the space bar is pressed). The alphanumeric 
   // characters (and in fact, all the characters) in the TIA Portal font have the peculiarity that they are
   // all a multiple of ⅓ of a normal space , the “i" for example is one normal space wide, “a” is 2⅓
   // normal space characters wide and “m” is 2⅔ normal space characters wide.
   // 
   // This “feature?” of the font is a distinct advantage; it means that is possible to always bring things
   // back into true alignment by using the range of whitespace characters. There are five such 
   // whitespace characters.
   // 
   // The width of the page is approximately 3.38 lowercase alphabets:
   // 
   // abcdefghijklmnopqrstuvwxyzabcdefghijklmnopqrstuvwxyzabcdefghijklmnopqrstuvwxyzabcdefghij
   // 
   // This averages at about 78 (non-space) characters per line.
   // 
   // A comment field can contain 65000 characters (approx.) including spaces and line breaks.
   // 
   // This broadly equates to 670 lines of standard text, approximately 13000 words.
   // 
   //                ━━━   ⬙⬙⬙⬙⬙⬙   ━━━
   // 
   // ██████████████ █ █ █ █  END   █ █ █ █ ██████████████
END_REGION

REGION Network 8: Example — Standard Tables
   // ▀▀▀▀▀▀▀▀▀▀▀▀▀▀▀▀▀▀▀▀▀▀▀▀▀▀▀▀▀▀▀▀▀▀▀▀▀▀▀▀▀▀▀▀
   // 
   // TITLE:    STANDARD TABLES (EXAMPLES)
   // 
   // ▄▄▄▄▄▄▄▄▄▄▄▄▄▄▄▄▄▄▄▄▄▄▄▄▄▄▄▄▄▄▄▄▄▄▄▄▄▄▄▄▄▄▄▄
   // 
   // 
   // 
   // Tables always have 2 blank lines above and 2 blank lines below.
   // 
   // ▌▌▌▌▌▌▌▌▌▌▌▌▌▌▌▌▌▌PARAMETER TABLE▐▐▐▐▐▐▐▐▐▐▐▐▐▐▐▐▐▐
   // 
   // 
   //  ――――――――――――――――――――――――――――――――――――――――――
   //  PARAM         FUNCTION                    TYPE      IN-OUT 
   //  ――――――――――――――――――――――――――――――――――――――――――
   //  SYS_SIGNALS      The system logic and timing signals for       UT21000    In
   //           parametric access
   // 
   //  RAW_ANALOG      The unscaled analogue input (input word         Word     In
   //           address for the IO card to which the instrument 
   //           is connected)
   // 
   //  RAW_MIN     Minimum value of the analogue input range      Int      In
   //           (see Table 3.1 to Table 3.3 for typical values)
   // 
   //  RAW_MAX       Maximum value of the analogue input range      Int      In
   //           (see Table 3.1 to Table 3.3 for typical values)
   // 
   //  SCALE_MIN    Calibrated lower value of the instrument       Real      In
   //           range in engineering units
   // 
   //  SCALE_MAX      Calibrated upper value of the instrument      Real      In
   //           range in engineering units
   // 
   //  STATIC_DATA     The static data associated with the PID loop       UT10001 In
   // 
   //  DYNAMIC_DATA      Stores the results of the event timing       UT38151    InOut
   //  ――――――――――――――――――――――――――――――――――――――――――
   // 
   // 
   // 
   // ▌▌▌▌▌▌▌▌▌▌▌▌▌▌▌▌▌ DATA STRUCTURE LIST ▐▐▐▐▐▐▐▐▐▐▐▐▐▐▐▐▐
   // 
   // 
   //  ――――――――――――――――――――――――――――――――――――――――――
   //  DATA STRUCTURE             DESCRIPTION
   //  ――――――――――――――――――――――――――――――――――――――――――
   //  UT01000_St_SysRevision          Revision information for this block    See FC01000
   //  UT01001_St_SysLicence           Licence information for this block  See FC01000
   //  UT21000_Dy_SysSignals           System signals for logic and timing  See FC01000
   // 
   //  UT02001_St_InstAnalogRead      Static data structure for an analogue instrument.
   //                     Holds configuration information, instrument ranges 
   //                     and scaling, alarm/warning thresholds &c.
   // 
   //  UT22001_Dy_InstAnalogRead        Dynamic data structure for an analogue instrument.
   //                     Current scaled instrument reading, alarm status, 
   //                     operating modes, timer values &c.
   //  ――――――――――――――――――――――――――――――――――――――――――
   // 
   // 
   // 
   // ▌▌▌▌▌▌▌▌▌▌   DATA STRUCTURE CONTENTS AND INSTANCE DBs   ▐▐▐▐▐▐▐▐▐▐
   // 
   // 
   //  UT38151_Dy_TimeEventRTC
   //  ――――――――――――――――――――――――――――――――――――――――――
   //  SIGNAL NAME          FUNCTION                     TYPE
   //  ――――――――――――――――――――――――――――――――――――――――――
   //  status_Running      STATUS — The event timer is running         Bool
   // 
   //  actual_StartTime      ACTUAL — Time at which the TRIGGER signal        DTL
   //                      went high (event start time)
   // 
   //  actual_EndTime        ACTUAL — Time at which the TRIGGER signal     DTL
   //                      went low (event end time)
   // 
   //  actual_Duration        ACTUAL — Event duration              LTime
   // 
   //  actual_DurationSec       ACTUAL — Event duration in seconds           REAL
   //  ――――――――――――――――――――――――――――――――――――――――――
   // 
   // 
   // 
   // 
   // ▌▌▌▌▌▌▌▌▌▌▌▌▌▌▌  CONSTANTS AND LOCAL DATA  ▐▐▐▐▐▐▐▐▐▐▐▐▐▐▐
   // 
   // [Keep local and constant data function description to one line and no gaps between rows]
   // 
   // 
   //  CONSTANTS DATA
   //  ――――――――――――――――――――――――――――――――――――――――――
   //  SIGNAL NAME          FUNCTION                     TYPE
   //  ――――――――――――――――――――――――――――――――――――――――――
   //  k_MIN_SP_HYST      Minimum value for SP achieved hysteresis (EU)     Real
   //  k_MIN_ALM_HYST      Minimum value for ALARM hysteresis (EU)       Real
   //  ――――――――――――――――――――――――――――――――――――――――――
   // 
   // 
   //  TEMPORARY (LOCAL) DATA
   //  ――――――――――――――――――――――――――――――――――――――――――
   //  SIGNAL NAME          FUNCTION                     TYPE
   //  ――――――――――――――――――――――――――――――――――――――――――
   //  wrkPercentPV          Process Variable as a percentage of inst. range     Real
   //  wrkPercentSP          Setpoint as a percentage of PV instrument range     Real
   //  wrkPercentDB         Deadband as a percentage of PV instrument range    Real
   //  wrkGain          Gain (adjusted for reverse/normal Acting)      Real
   //  wrkCycTime          Cyclic execution time (TIME format)         Time
   //  ――――――――――――――――――――――――――――――――――――――――――
   // 
   // 
   // 
   // ▌▌▌▌▌▌▌▌▌▌▌▌▌▌▌▌▌▌▌  BLOCK LIST  ▐▐▐▐▐▐▐▐▐▐▐▐▐▐▐▐▐▐▐
   // 
   // 
   //  BLOCK CALLS
   //  ――――――――――――――――――――――――――――――――――――――――――
   //  BLOCK          TITLE             DESCRIPTION  
   //  ――――――――――――――――――――――――――――――――――――――――――
   //  FC18001         StdSubScaleAI        Scales an analogue input signal 
   //                            Continuation line
   //  ――――――――――――――――――――――――――――――――――――――――――
   // 
   // 
   //  ASSOCIATED BLOCKS
   //  ――――――――――――――――――――――――――――――――――――――――――
   //  BLOCK          TITLE             DESCRIPTION  
   //  ――――――――――――――――――――――――――――――――――――――――――
   //  FC17102         StdCommsWrite65K       Write data partner block
   //                            Continuation line 
   //  ――――――――――――――――――――――――――――――――――――――――――
   // 
   // 
   // 
   // ▌▌▌▌▌▌▌▌▌▌▌▌▌▌▌▌▌  SYSTEM BLOCK LIST   ▐▐▐▐▐▐▐▐▐▐▐▐▐▐▐▐▐
   // 
   // 
   //  SYSTEM BLOCK CALLS
   //  ――――――――――――――――――――――――――――――――――――――――――
   //  BLOCK          TITLE             DESCRIPTION  
   //  ――――――――――――――――――――――――――――――――――――――――――
   //  RD_LOC_T             Read the local RTC time    Reads the CPU real time clock 
   //  (FC804)                        Continuation line 
   //                            Continuation line
   //  ――――――――――――――――――――――――――――――――――――――――――
   // 
   // 
   // ▌▌▌▌▌▌▌▌▌▌▌▌▌▌▌▌▌▌▌▌▌▌▐▐▐▐▐▐▐▐▐▐▐▐▐▐▐▐▐▐▐▐▐▐
   // 
   // 
   //                ━━━   ⬙⬙⬙⬙⬙⬙   ━━━
   // 
   // 
   // ██████████████ █ █ █ █  END   █ █ █ █ ██████████████
END_REGION

REGION Network 9: Example — Other tables
   // ▀▀▀▀▀▀▀▀▀▀▀▀▀▀▀▀▀▀▀▀▀▀▀▀▀▀▀▀▀▀▀▀▀▀▀▀▀▀▀▀▀▀▀▀
   // 
   // TITLE:    OTHER TABLES (EXAMPLES)
   // 
   // ▄▄▄▄▄▄▄▄▄▄▄▄▄▄▄▄▄▄▄▄▄▄▄▄▄▄▄▄▄▄▄▄▄▄▄▄▄▄▄▄▄▄▄▄
   // 
   // 
   // 
   // Tables always have 2 blank lines above and 2 blank lines below.
   // 
   // 
   // ▌▌▌▌▌▌▌▌▌▌▌▌▌▌▌▌▌  TWO COLUMN TABLE ▐▐▐▐▐▐▐▐▐▐▐▐▐▐▐▐▐
   // 
   // 
   //  ――――――――――――――――――――――――――――――――――――――――――
   //  IO TYPE            DESCRIPTION
   //  ――――――――――――――――――――――――――――――――――――――――――
   //  ET200MP         Standard IO high density IO for the S7-1500 range
   // 
   //  ET200M           Standard IO high density IO for the S7-300 range, 
   //               can be used as remote IO for the S7-1500
   //  ――――――――――――――――――――――――――――――――――――――――――
   // 
   // 
   // ▌▌▌▌▌▌▌▌▌▌▌▌▌▌▌▌▌THREE COLUMN TABLE ▐▐▐▐▐▐▐▐▐▐▐▐▐▐▐▐▐
   // 
   // [Numerical table with number alignment to the right]
   // 
   // 
   //  ――――――――――――――――――――――――――――――――――――――――――
   //  PRESSURE           RAW SIGNAL           SCALED VAL
   //  ――――――――――――――――――――――――――――――――――――――――――
   //  -250.0 Pa                   0             -250.0 Pa
   //        0.0 Pa                  13824            0.0 Pa
   //   250.0 Pa                  27648              250.0 Pa
   //  ――――――――――――――――――――――――――――――――――――――――――
   // 
   // 
   // ▌▌▌▌▌▌▌▌▌▌▌▌▌▌▌▌▌ FOUR COLUMN TABLE ▐▐▐▐▐▐▐▐▐▐▐▐▐▐▐▐▐
   // 
   // [Numerical table with number alignment to the right]
   // 
   // 
   //  ――――――――――――――――――――――――――――――――――――――――――
   //  RAW MIN       RAW MAX      SCALED MIN       SCALED MAX
   //  ――――――――――――――――――――――――――――――――――――――――――
   //        0        27648        -250.0 Pa        250.0 Pa
   //  ――――――――――――――――――――――――――――――――――――――――――
   // 
   // 
   // ▌▌▌▌▌▌▌▌▌▌▌▌▌▌▌▌▌  TABLE WITH HEADING  ▐▐▐▐▐▐▐▐▐▐▐▐▐▐▐▐▐
   // 
   // [Numerical table with number alignment to the right]
   // 
   // 
   //  CURRENT SIGNALS
   //  ――――――――――――――――――――――――――――――――――――――――――
   //  SIGNAL TYPE     SIG MIN VAL      RAW_MIN     SIG MAX VAL     RAW_MAX
   //  ――――――――――――――――――――――――――――――――――――――――――
   //    4-20 mA      4 mA          0          20 mA       27648
   //    0-20 mA      0 mA          0          20 mA       27648
   //  -20 to 20 mA      -20 mA      -27648          20 mA       27648
   //  ――――――――――――――――――――――――――――――――――――――――――
   // 
   // 
   // 
   // ▌▌▌▌▌▌▌▌▌▌▌▌▌▌▌▌▌▌▌▌▌▌▐▐▐▐▐▐▐▐▐▐▐▐▐▐▐▐▐▐▐▐▐▐
   // 
   //                ━━━   ⬙⬙⬙⬙⬙⬙   ━━━
   // 
   // 
   // ██████████████ █ █ █ █  END   █ █ █ █ ██████████████
END_REGION

